LIN {X 0,Y 468.05,Z 517.764,A -85,B 0,C 180,E1 -7638.744,E2 -7638.744} C_VEL
LIN {X 0,Y 467.575,Z 526.244,A -85,B 0,C 180,E1 -7639.828,E2 -7639.828} C_VEL
LIN {X 0,Y 467.241,Z 534.525,A -85,B 0,C 180,E1 -7641.131,E2 -7641.131} C_VEL
LIN {X 0,Y 466.979,Z 541.203,A -85,B 0,C 180,E1 -7642.433,E2 -7642.433} C_VEL
LIN {X 0,Y 466.773,Z 547.316,A -85,B 0,C 180,E1 -7643.95,E2 -7643.95} C_VEL
LIN {X 0,Y 466.694,Z 551.29,A -85,B 0,C 180,E1 -7645.249,E2 -7645.249} C_VEL
LIN {X 0,Y 466.691,Z 554.227,A -85,B 0,C 180,E1 -7646.546,E2 -7646.546} C_VEL
LIN {X 0,Y 466.662,Z 555.625,A -85,B 0,C 180,E1 -7647.41,E2 -7647.41} C_VEL
LIN {X 0,Y 466.618,Z 557.234,A -85,B 0,C 180,E1 -7649.137,E2 -7649.137} C_VEL
LIN {X 0,Y 466.598,Z 557.451,A -85,B 0,C 180,E1 -7650,E2 -7650} C_VEL
LIN {X 0,Y 466.618,Z 557.236,A -85,B 0,C 180,E1 -7650.863,E2 -7650.863} C_VEL
LIN {X 0,Y 466.662,Z 555.636,A -85,B 0,C 180,E1 -7652.589,E2 -7652.589} C_VEL
LIN {X 0,Y 466.691,Z 554.239,A -85,B 0,C 180,E1 -7653.453,E2 -7653.453} C_VEL
LIN {X 0,Y 466.694,Z 551.3,A -85,B 0,C 180,E1 -7654.751,E2 -7654.751} C_VEL
LIN {X 0,Y 466.778,Z 547.322,A -85,B 0,C 180,E1 -7656.05,E2 -7656.05} C_VEL
LIN {X 0,Y 466.979,Z 541.2,A -85,B 0,C 180,E1 -7657.567,E2 -7657.567} C_VEL
LIN {X 0,Y 467.24,Z 534.511,A -85,B 0,C 180,E1 -7658.869,E2 -7658.869} C_VEL
LIN {X 0,Y 467.586,Z 526.211,A -85,B 0,C 180,E1 -7660.172,E2 -7660.172} C_VEL
LIN {X 0,Y 468.04,Z 517.699,A -85,B 0,C 180,E1 -7661.256,E2 -7661.256} C_VEL
LIN {X 0,Y 468.53,Z 507.566,A -85,B 0,C 180,E1 -7662.306,E2 -7662.306} C_VEL
LIN {X 0,Y 468.963,Z 496.77,A -85,B 0,C 180,E1 -7663.211,E2 -7663.211} C_VEL
LIN {X 0,Y 469.508,Z 485.356,A -85,B 0,C 180,E1 -7663.967,E2 -7663.967} C_VEL
LIN {X 0,Y 469.937,Z 473.595,A -85,B 0,C 180,E1 -7664.562,E2 -7664.562} C_VEL
LIN {X 0,Y 469.738,Z 468.411,A -85,B 0,C 180,E1 -7664.783,E2 -7664.783} C_VEL
LIN {X 0,Y 467.641,Z 455.017,A -85,B 0,C 180,E1 -7665.263,E2 -7665.263} C_VEL
LIN {X 0,Y 466.967,Z 450.66,A -85,B 0,C 180,E1 -7665.391,E2 -7665.391} C_VEL
LIN {X 0,Y 467.115,Z 442.772,A -85,B 0,C 180,E1 -7668.581,E2 -7668.581} C_VEL
LIN {X 0,Y 467.351,Z 435.39,A -85,B 0,C 180,E1 -7671.618,E2 -7671.618} C_VEL
LIN {X 0,Y 467.538,Z 427.589,A -85,B 0,C 180,E1 -7674.89,E2 -7674.89} C_VEL
LIN {X 0,Y 467.819,Z 419.776,A -85,B 0,C 180,E1 -7678.243,E2 -7678.243} C_VEL
LIN {X 0,Y 468.09,Z 413.208,A -85,B 0,C 180,E1 -7681.15,E2 -7681.15} C_VEL
LIN {X 0,Y 468.397,Z 406.109,A -85,B 0,C 180,E1 -7684.387,E2 -7684.387} C_VEL
LIN {X 0,Y 468.342,Z 401.978,A -85,B 0,C 180,E1 -7686.35,E2 -7686.35} C_VEL
LIN {X 0,Y 467.644,Z 397.237,A -85,B 0,C 180,E1 -7688.752,E2 -7688.752} C_VEL
LIN {X 0,Y 467.579,Z 397.243,A -85,B 0,C 180,E1 -7691.401,E2 -7691.401} C_VEL
LIN {X 0,Y 467.57,Z 397.24,A -85,B 0,C 180,E1 -7693.823,E2 -7693.823} C_VEL
LIN {X 0,Y 467.565,Z 397.242,A -85,B 0,C 180,E1 -7696.256,E2 -7696.256} C_VEL
LIN {X 0,Y 467.577,Z 397.244,A -85,B 0,C 180,E1 -7698.722,E2 -7698.722} C_VEL
LIN {X 0,Y 467.561,Z 397.242,A -85,B 0,C 180,E1 -7701.955,E2 -7701.955} C_VEL
LIN {X 0,Y 467.563,Z 397.242,A -85,B 0,C 180,E1 -7705.167,E2 -7705.167} C_VEL
LIN {X 0,Y 467.579,Z 397.242,A -85,B 0,C 180,E1 -7708.259,E2 -7708.259} C_VEL
LIN {X 0,Y 467.576,Z 397.24,A -85,B 0,C 180,E1 -7711.25,E2 -7711.25} C_VEL
LIN {X 0,Y 467.603,Z 397.239,A -85,B 0,C 180,E1 -7714.159,E2 -7714.159} C_VEL
LIN {X 0,Y 467.57,Z 397.241,A -85,B 0,C 180,E1 -7716.995,E2 -7716.995} C_VEL
LIN {X 0,Y 467.614,Z 397.237,A -85,B 0,C 180,E1 -7719.777,E2 -7719.777} C_VEL
LIN {X 0,Y 467.601,Z 397.238,A -85,B 0,C 180,E1 -7722.506,E2 -7722.506} C_VEL
LIN {X 0,Y 467.598,Z 397.239,A -85,B 0,C 180,E1 -7725.196,E2 -7725.196} C_VEL
LIN {X 0,Y 467.647,Z 397.234,A -85,B 0,C 180,E1 -7727.854,E2 -7727.854} C_VEL
LIN {X 0,Y 467.673,Z 397.23,A -85,B 0,C 180,E1 -7731.357,E2 -7731.357} C_VEL
LIN {X 0,Y 467.739,Z 397.222,A -85,B 0,C 180,E1 -7733.962,E2 -7733.962} C_VEL
LIN {X 0,Y 467.852,Z 397.208,A -85,B 0,C 180,E1 -7737.417,E2 -7737.417} C_VEL
LIN {X 0,Y 467.873,Z 397.204,A -85,B 0,C 180,E1 -7740,E2 -7740} C_VEL
LIN {X 0,Y 467.853,Z 397.207,A -85,B 0,C 180,E1 -7742.583,E2 -7742.583} C_VEL
LIN {X 0,Y 467.739,Z 397.22,A -85,B 0,C 180,E1 -7746.037,E2 -7746.037} C_VEL
LIN {X 0,Y 467.674,Z 397.232,A -85,B 0,C 180,E1 -7748.643,E2 -7748.643} C_VEL
LIN {X 0,Y 467.656,Z 397.231,A -85,B 0,C 180,E1 -7752.145,E2 -7752.145} C_VEL
LIN {X 0,Y 467.63,Z 397.233,A -85,B 0,C 180,E1 -7755.695,E2 -7755.695} C_VEL
LIN {X 0,Y 467.609,Z 397.238,A -85,B 0,C 180,E1 -7758.765,E2 -7758.765} C_VEL
LIN {X 0,Y 467.575,Z 397.24,A -85,B 0,C 180,E1 -7761.27,E2 -7761.27} C_VEL
LIN {X 0,Y 467.567,Z 397.243,A -85,B 0,C 180,E1 -7763.943,E2 -7763.943} C_VEL
LIN {X 0,Y 467.62,Z 397.235,A -85,B 0,C 180,E1 -7766.8,E2 -7766.8} C_VEL
LIN {X 0,Y 467.58,Z 397.241,A -85,B 0,C 180,E1 -7769.736,E2 -7769.736} C_VEL
LIN {X 0,Y 467.576,Z 397.24,A -85,B 0,C 180,E1 -7772.759,E2 -7772.759} C_VEL
LIN {X 0,Y 467.55,Z 397.248,A -85,B 0,C 180,E1 -7775.89,E2 -7775.89} C_VEL
LIN {X 0,Y 467.612,Z 397.235,A -85,B 0,C 180,E1 -7779.142,E2 -7779.142} C_VEL
LIN {X 0,Y 467.613,Z 397.234,A -85,B 0,C 180,E1 -7782.572,E2 -7782.572} C_VEL
LIN {X 0,Y 467.569,Z 397.24,A -85,B 0,C 180,E1 -7786.177,E2 -7786.177} C_VEL
LIN {X 0,Y 467.585,Z 397.237,A -85,B 0,C 180,E1 -7788.722,E2 -7788.722} C_VEL
LIN {X 0,Y 467.57,Z 397.245,A -85,B 0,C 180,E1 -7791.408,E2 -7791.408} C_VEL
LIN {X 0,Y 467.56,Z 397.239,A -85,B 0,C 180,E1 -7794.261,E2 -7794.261} C_VEL
LIN {X 0,Y 467.579,Z 397.245,A -85,B 0,C 180,E1 -7797.321,E2 -7797.321} C_VEL
LIN {X 0,Y 467.568,Z 397.241,A -85,B 0,C 180,E1 -7800.668,E2 -7800.668} C_VEL
LIN {X 0,Y 467.626,Z 397.238,A -85,B 0,C 180,E1 -7803.201,E2 -7803.201} C_VEL
LIN {X 0,Y 467.591,Z 397.238,A -85,B 0,C 180,E1 -7806.469,E2 -7806.469} C_VEL
LIN {X 0,Y 467.461,Z 397.258,A -85,B 0,C 180,E1 -7808.85,E2 -7808.85} C_VEL
LIN {X 0,Y 467.399,Z 398.142,A -85,B 0,C 180,E1 -7809.768,E2 -7809.768} C_VEL
LIN {X 0,Y 467.349,Z 402.042,A -85,B 0,C 180,E1 -7812.497,E2 -7812.497} C_VEL
LIN {X 0,Y 467.262,Z 406.123,A -85,B 0,C 180,E1 -7815.305,E2 -7815.305} C_VEL
LIN {X 0,Y 466.552,Z 407.238,A -85,B 0,C 180,E1 -7816.012,E2 -7816.012} C_VEL
LIN {X 0,Y 463.68,Z 409.212,A -85,B 0,C 180,E1 -7817.157,E2 -7817.157} C_VEL
LIN {X 0,Y 461.256,Z 410.811,A -85,B 0,C 180,E1 -7818.079,E2 -7818.079} C_VEL
LIN {X 0,Y 460.19,Z 411.965,A -85,B 0,C 180,E1 -7818.793,E2 -7818.793} C_VEL
LIN {X 0,Y 460.088,Z 412.332,A -85,B 0,C 180,E1 -7819.035,E2 -7819.035} C_VEL
LIN {X 0,Y 460,Z 416.903,A -85,B 0,C 180,E1 -7822.097,E2 -7822.097} C_VEL
LIN {X 0,Y 460.007,Z 419.564,A -85,B 0,C 180,E1 -7823.861,E2 -7823.861} C_VEL
LIN {X 0,Y 459.953,Z 423.574,A -85,B 0,C 180,E1 -7826.496,E2 -7826.496} C_VEL
LIN {X 0,Y 459.695,Z 426.637,A -85,B 0,C 180,E1 -7828.467,E2 -7828.467} C_VEL
LIN {X 0,Y 462.589,Z 440.592,A -85,B 0,C 180,E1 -7828.98,E2 -7828.98} C_VEL
LIN {X 0,Y 463.245,Z 445.212,A -85,B 0,C 180,E1 -7829.185,E2 -7829.185} C_VEL
LIN {X 0,Y 462.884,Z 457.387,A -85,B 0,C 180,E1 -7829.783,E2 -7829.783} C_VEL
LIN {X 0,Y 462.302,Z 469.202,A -85,B 0,C 180,E1 -7830.545,E2 -7830.545} C_VEL
LIN {X 0,Y 461.851,Z 479.727,A -85,B 0,C 180,E1 -7831.417,E2 -7831.417} C_VEL
LIN {X 0,Y 461.333,Z 489.381,A -85,B 0,C 180,E1 -7832.401,E2 -7832.401} C_VEL
LIN {X 0,Y 460.819,Z 498.195,A -85,B 0,C 180,E1 -7833.498,E2 -7833.498} C_VEL
LIN {X 0,Y 460.377,Z 506.8,A -85,B 0,C 180,E1 -7834.816,E2 -7834.816} C_VEL
LIN {X 0,Y 460.156,Z 513.662,A -85,B 0,C 180,E1 -7836.137,E2 -7836.137} C_VEL
LIN {X 0,Y 459.923,Z 519.186,A -85,B 0,C 180,E1 -7837.463,E2 -7837.463} C_VEL
LIN {X 0,Y 459.711,Z 523.535,A -85,B 0,C 180,E1 -7838.794,E2 -7838.794} C_VEL
LIN {X 0,Y 459.612,Z 525.839,A -85,B 0,C 180,E1 -7839.683,E2 -7839.683} C_VEL
LIN {X 0,Y 459.606,Z 527.696,A -85,B 0,C 180,E1 -7840.573,E2 -7840.573} C_VEL
LIN {X 0,Y 459.566,Z 529.559,A -85,B 0,C 180,E1 -7841.838,E2 -7841.838} C_VEL
LIN {X 0,Y 459.439,Z 530.67,A -85,B 0,C 180,E1 -7843.265,E2 -7843.265} C_VEL
LIN {X 0,Y 459.437,Z 530.824,A -85,B 0,C 180,E1 -7844.167,E2 -7844.167} C_VEL
LIN {X 0,Y 459.496,Z 530.297,A -85,B 0,C 180,E1 -7845.51,E2 -7845.51} C_VEL
LIN {X 0,Y 459.465,Z 528.774,A -85,B 0,C 180,E1 -7846.895,E2 -7846.895} C_VEL
LIN {X 0,Y 459.645,Z 525.549,A -85,B 0,C 180,E1 -7848.561,E2 -7848.561} C_VEL
LIN {X 0,Y 459.816,Z 521.139,A -85,B 0,C 180,E1 -7850.114,E2 -7850.114} C_VEL
LIN {X 0,Y 460.065,Z 515.868,A -85,B 0,C 180,E1 -7851.507,E2 -7851.507} C_VEL
LIN {X 0,Y 460.391,Z 509.082,A -85,B 0,C 180,E1 -7852.908,E2 -7852.908} C_VEL
LIN {X 0,Y 460.803,Z 500.493,A -85,B 0,C 180,E1 -7854.317,E2 -7854.317} C_VEL
LIN {X 0,Y 461.28,Z 491.756,A -85,B 0,C 180,E1 -7855.473,E2 -7855.473} C_VEL
LIN {X 0,Y 461.797,Z 481.616,A -85,B 0,C 180,E1 -7856.554,E2 -7856.554} C_VEL
LIN {X 0,Y 462.412,Z 470.625,A -85,B 0,C 180,E1 -7857.494,E2 -7857.494} C_VEL
LIN {X 0,Y 462.852,Z 460.595,A -85,B 0,C 180,E1 -7858.181,E2 -7858.181} C_VEL
LIN {X 0,Y 463.292,Z 448.73,A -85,B 0,C 180,E1 -7858.817,E2 -7858.817} C_VEL
LIN {X 0,Y 463.261,Z 443.626,A -85,B 0,C 180,E1 -7859.042,E2 -7859.042} C_VEL
LIN {X 0,Y 460.731,Z 431.182,A -85,B 0,C 180,E1 -7859.558,E2 -7859.558} C_VEL
LIN {X 0,Y 459.714,Z 426.771,A -85,B 0,C 180,E1 -7859.711,E2 -7859.711} C_VEL
LIN {X 0,Y 459.836,Z 422.121,A -85,B 0,C 180,E1 -7862.796,E2 -7862.796} C_VEL
LIN {X 0,Y 459.944,Z 417.5,A -85,B 0,C 180,E1 -7865.919,E2 -7865.919} C_VEL
LIN {X 0,Y 460.079,Z 413.289,A -85,B 0,C 180,E1 -7868.826,E2 -7868.826} C_VEL
LIN {X 0,Y 460.181,Z 409.438,A -85,B 0,C 180,E1 -7871.553,E2 -7871.553} C_VEL
LIN {X 0,Y 460.298,Z 405.231,A -85,B 0,C 180,E1 -7874.615,E2 -7874.615} C_VEL
LIN {X 0,Y 460.461,Z 400.928,A -85,B 0,C 180,E1 -7877.812,E2 -7877.812} C_VEL
LIN {X 0,Y 460.444,Z 398.134,A -85,B 0,C 180,E1 -7880.129,E2 -7880.129} C_VEL
LIN {X 0,Y 460.496,Z 398.129,A -85,B 0,C 180,E1 -7882.523,E2 -7882.523} C_VEL
LIN {X 0,Y 460.543,Z 398.121,A -85,B 0,C 180,E1 -7885.624,E2 -7885.624} C_VEL
LIN {X 0,Y 460.531,Z 398.12,A -85,B 0,C 180,E1 -7888.744,E2 -7888.744} C_VEL
LIN {X 0,Y 460.553,Z 398.117,A -85,B 0,C 180,E1 -7891.767,E2 -7891.767} C_VEL
LIN {X 0,Y 460.554,Z 398.117,A -85,B 0,C 180,E1 -7894.705,E2 -7894.705} C_VEL
LIN {X 0,Y 460.505,Z 398.122,A -85,B 0,C 180,E1 -7897.571,E2 -7897.571} C_VEL
LIN {X 0,Y 460.562,Z 398.116,A -85,B 0,C 180,E1 -7900.384,E2 -7900.384} C_VEL
LIN {X 0,Y 460.559,Z 398.117,A -85,B 0,C 180,E1 -7903.146,E2 -7903.146} C_VEL
LIN {X 0,Y 460.548,Z 398.118,A -85,B 0,C 180,E1 -7905.868,E2 -7905.868} C_VEL
LIN {X 0,Y 460.607,Z 398.109,A -85,B 0,C 180,E1 -7908.559,E2 -7908.559} C_VEL
LIN {X 0,Y 460.688,Z 398.103,A -85,B 0,C 180,E1 -7912.109,E2 -7912.109} C_VEL
LIN {X 0,Y 460.691,Z 398.1,A -85,B 0,C 180,E1 -7914.748,E2 -7914.748} C_VEL
LIN {X 0,Y 460.819,Z 398.082,A -85,B 0,C 180,E1 -7917.378,E2 -7917.378} C_VEL
LIN {X 0,Y 460.846,Z 398.08,A -85,B 0,C 180,E1 -7920,E2 -7920} C_VEL
LIN {X 0,Y 460.819,Z 398.086,A -85,B 0,C 180,E1 -7922.623,E2 -7922.623} C_VEL
LIN {X 0,Y 460.704,Z 398.097,A -85,B 0,C 180,E1 -7926.13,E2 -7926.13} C_VEL
LIN {X 0,Y 460.623,Z 398.109,A -85,B 0,C 180,E1 -7928.776,E2 -7928.776} C_VEL
LIN {X 0,Y 460.628,Z 398.107,A -85,B 0,C 180,E1 -7932.457,E2 -7932.457} C_VEL
LIN {X 0,Y 460.616,Z 398.113,A -85,B 0,C 180,E1 -7936.008,E2 -7936.008} C_VEL
LIN {X 0,Y 460.564,Z 398.116,A -85,B 0,C 180,E1 -7939.616,E2 -7939.616} C_VEL
LIN {X 0,Y 460.507,Z 398.124,A -85,B 0,C 180,E1 -7942.429,E2 -7942.429} C_VEL
LIN {X 0,Y 460.564,Z 398.116,A -85,B 0,C 180,E1 -7945.803,E2 -7945.803} C_VEL
LIN {X 0,Y 460.554,Z 398.118,A -85,B 0,C 180,E1 -7948.233,E2 -7948.233} C_VEL
LIN {X 0,Y 460.521,Z 398.122,A -85,B 0,C 180,E1 -7951.284,E2 -7951.284} C_VEL
LIN {X 0,Y 460.53,Z 398.119,A -85,B 0,C 180,E1 -7954.507,E2 -7954.507} C_VEL
LIN {X 0,Y 460.525,Z 398.116,A -85,B 0,C 180,E1 -7957.621,E2 -7957.621} C_VEL
LIN {X 0,Y 460.539,Z 398.119,A -85,B 0,C 180,E1 -7960.27,E2 -7960.27} C_VEL
LIN {X 0,Y 460.498,Z 398.125,A -85,B 0,C 180,E1 -7963.376,E2 -7963.376} C_VEL
LIN {X 0,Y 460.507,Z 398.123,A -85,B 0,C 180,E1 -7966.626,E2 -7966.626} C_VEL
LIN {X 0,Y 460.556,Z 398.119,A -85,B 0,C 180,E1 -7969.937,E2 -7969.937} C_VEL
LIN {X 0,Y 461.273,Z 402.381,A -85,B 0,C 180,E1 -7972.451,E2 -7972.451} C_VEL
LIN {X 0,Y 461.655,Z 406.549,A -85,B 0,C 180,E1 -7974.656,E2 -7974.656} C_VEL
LIN {X 0,Y 461.413,Z 411.029,A -85,B 0,C 180,E1 -7976.902,E2 -7976.902} C_VEL
LIN {X 0,Y 461.136,Z 417.074,A -85,B 0,C 180,E1 -7979.806,E2 -7979.806} C_VEL
LIN {X 0,Y 460.713,Z 423.504,A -85,B 0,C 180,E1 -7982.766,E2 -7982.766} C_VEL
LIN {X 0,Y 460.467,Z 429.999,A -85,B 0,C 180,E1 -7985.664,E2 -7985.664} C_VEL
LIN {X 0,Y 460.277,Z 436.882,A -85,B 0,C 180,E1 -7988.657,E2 -7988.657} C_VEL
LIN {X 0,Y 460.03,Z 444.198,A -85,B 0,C 180,E1 -7991.749,E2 -7991.749} C_VEL
LIN {X 0,Y 459.886,Z 450.374,A -85,B 0,C 180,E1 -7994.317,E2 -7994.317} C_VEL
LIN {X 0,Y 462.057,Z 463.442,A -85,B 0,C 180,E1 -7994.748,E2 -7994.748} C_VEL
LIN {X 0,Y 463.163,Z 472.924,A -85,B 0,C 180,E1 -7995.164,E2 -7995.164} C_VEL
LIN {X 0,Y 462.724,Z 483.778,A -85,B 0,C 180,E1 -7995.711,E2 -7995.711} C_VEL
LIN {X 0,Y 462.174,Z 495.488,A -85,B 0,C 180,E1 -7996.479,E2 -7996.479} C_VEL
LIN {X 0,Y 461.704,Z 505.916,A -85,B 0,C 180,E1 -7997.348,E2 -7997.348} C_VEL
LIN {X 0,Y 461.199,Z 515.71,A -85,B 0,C 180,E1 -7998.351,E2 -7998.351} C_VEL
LIN {X 0,Y 460.622,Z 524.523,A -85,B 0,C 180,E1 -7999.45,E2 -7999.45} C_VEL
LIN {X 0,Y 460.241,Z 533.123,A -85,B 0,C 180,E1 -8000.774,E2 -8000.774} C_VEL
LIN {X 0,Y 459.952,Z 540.009,A -85,B 0,C 180,E1 -8002.096,E2 -8002.096} C_VEL
LIN {X 0,Y 459.715,Z 546.095,A -85,B 0,C 180,E1 -8003.569,E2 -8003.569} C_VEL
LIN {X 0,Y 459.622,Z 551.095,A -85,B 0,C 180,E1 -8005.176,E2 -8005.176} C_VEL
LIN {X 0,Y 459.586,Z 554.03,A -85,B 0,C 180,E1 -8006.493,E2 -8006.493} C_VEL
LIN {X 0,Y 459.585,Z 555.426,A -85,B 0,C 180,E1 -8007.37,E2 -8007.37} C_VEL
LIN {X 0,Y 459.522,Z 557.032,A -85,B 0,C 180,E1 -8009.124,E2 -8009.124} C_VEL
LIN {X 0,Y 459.53,Z 557.248,A -85,B 0,C 180,E1 -8010,E2 -8010} C_VEL
LIN {X 0,Y 459.521,Z 557.03,A -85,B 0,C 180,E1 -8010.876,E2 -8010.876} C_VEL
LIN {X 0,Y 459.585,Z 555.427,A -85,B 0,C 180,E1 -8012.629,E2 -8012.629} C_VEL
LIN {X 0,Y 459.586,Z 554.026,A -85,B 0,C 180,E1 -8013.507,E2 -8013.507} C_VEL
LIN {X 0,Y 459.622,Z 551.085,A -85,B 0,C 180,E1 -8014.824,E2 -8014.824} C_VEL
LIN {X 0,Y 459.714,Z 546.066,A -85,B 0,C 180,E1 -8016.431,E2 -8016.431} C_VEL
LIN {X 0,Y 459.951,Z 539.96,A -85,B 0,C 180,E1 -8017.904,E2 -8017.904} C_VEL
LIN {X 0,Y 460.24,Z 533.036,A -85,B 0,C 180,E1 -8019.226,E2 -8019.226} C_VEL
LIN {X 0,Y 460.629,Z 524.356,A -85,B 0,C 180,E1 -8020.549,E2 -8020.549} C_VEL
LIN {X 0,Y 461.137,Z 515.46,A -85,B 0,C 180,E1 -8021.65,E2 -8021.65} C_VEL
LIN {X 0,Y 461.686,Z 505.699,A -85,B 0,C 180,E1 -8022.639,E2 -8022.639} C_VEL
LIN {X 0,Y 462.133,Z 494.977,A -85,B 0,C 180,E1 -8023.522,E2 -8023.522} C_VEL
LIN {X 0,Y 462.646,Z 482.967,A -85,B 0,C 180,E1 -8024.291,E2 -8024.291} C_VEL
LIN {X 0,Y 463.091,Z 471.765,A -85,B 0,C 180,E1 -8024.838,E2 -8024.838} C_VEL
LIN {X 0,Y 461.183,Z 458.423,A -85,B 0,C 180,E1 -8025.376,E2 -8025.376} C_VEL
LIN {X 0,Y 459.881,Z 450.497,A -85,B 0,C 180,E1 -8025.612,E2 -8025.612} C_VEL
LIN {X 0,Y 460.053,Z 442.965,A -85,B 0,C 180,E1 -8028.711,E2 -8028.711} C_VEL
LIN {X 0,Y 460.301,Z 435.181,A -85,B 0,C 180,E1 -8031.966,E2 -8031.966} C_VEL
LIN {X 0,Y 460.523,Z 427.377,A -85,B 0,C 180,E1 -8035.296,E2 -8035.296} C_VEL
LIN {X 0,Y 460.837,Z 419.593,A -85,B 0,C 180,E1 -8038.71,E2 -8038.71} C_VEL
LIN {X 0,Y 461.094,Z 413.614,A -85,B 0,C 180,E1 -8041.399,E2 -8041.399} C_VEL
LIN {X 0,Y 461.399,Z 406.578,A -85,B 0,C 180,E1 -8044.661,E2 -8044.661} C_VEL
LIN {X 0,Y 461.297,Z 402.887,A -85,B 0,C 180,E1 -8046.453,E2 -8046.453} C_VEL
LIN {X 0,Y 460.604,Z 398.114,A -85,B 0,C 180,E1 -8048.906,E2 -8048.906} C_VEL
LIN {X 0,Y 460.523,Z 398.12,A -85,B 0,C 180,E1 -8052.18,E2 -8052.18} C_VEL
LIN {X 0,Y 460.517,Z 398.12,A -85,B 0,C 180,E1 -8055.411,E2 -8055.411} C_VEL
LIN {X 0,Y 460.53,Z 398.119,A -85,B 0,C 180,E1 -8058.396,E2 -8058.396} C_VEL
LIN {X 0,Y 460.521,Z 398.119,A -85,B 0,C 180,E1 -8061.266,E2 -8061.266} C_VEL
LIN {X 0,Y 460.508,Z 398.124,A -85,B 0,C 180,E1 -8064.554,E2 -8064.554} C_VEL
LIN {X 0,Y 460.526,Z 398.119,A -85,B 0,C 180,E1 -8067.715,E2 -8067.715} C_VEL
LIN {X 0,Y 460.541,Z 398.119,A -85,B 0,C 180,E1 -8070.769,E2 -8070.769} C_VEL
LIN {X 0,Y 460.556,Z 398.116,A -85,B 0,C 180,E1 -8073.734,E2 -8073.734} C_VEL
LIN {X 0,Y 460.539,Z 398.119,A -85,B 0,C 180,E1 -8076.623,E2 -8076.623} C_VEL
LIN {X 0,Y 460.543,Z 398.118,A -85,B 0,C 180,E1 -8079.452,E2 -8079.452} C_VEL
LIN {X 0,Y 460.551,Z 398.119,A -85,B 0,C 180,E1 -8082.23,E2 -8082.23} C_VEL
LIN {X 0,Y 460.557,Z 398.115,A -85,B 0,C 180,E1 -8084.964,E2 -8084.964} C_VEL
LIN {X 0,Y 460.602,Z 398.109,A -85,B 0,C 180,E1 -8088.559,E2 -8088.559} C_VEL
LIN {X 0,Y 460.686,Z 398.1,A -85,B 0,C 180,E1 -8092.108,E2 -8092.108} C_VEL
LIN {X 0,Y 460.694,Z 398.099,A -85,B 0,C 180,E1 -8094.748,E2 -8094.748} C_VEL
LIN {X 0,Y 460.817,Z 398.084,A -85,B 0,C 180,E1 -8097.377,E2 -8097.377} C_VEL
LIN {X 0,Y 460.844,Z 398.08,A -85,B 0,C 180,E1 -8100,E2 -8100} C_VEL
LIN {X 0,Y 460.818,Z 398.084,A -85,B 0,C 180,E1 -8102.622,E2 -8102.622} C_VEL
LIN {X 0,Y 460.704,Z 398.097,A -85,B 0,C 180,E1 -8106.13,E2 -8106.13} C_VEL
LIN {X 0,Y 460.621,Z 398.11,A -85,B 0,C 180,E1 -8108.776,E2 -8108.776} C_VEL
LIN {X 0,Y 460.625,Z 398.109,A -85,B 0,C 180,E1 -8112.457,E2 -8112.457} C_VEL
LIN {X 0,Y 460.591,Z 398.111,A -85,B 0,C 180,E1 -8115.998,E2 -8115.998} C_VEL
LIN {X 0,Y 460.562,Z 398.115,A -85,B 0,C 180,E1 -8118.902,E2 -8118.902} C_VEL
LIN {X 0,Y 460.51,Z 398.12,A -85,B 0,C 180,E1 -8121.486,E2 -8121.486} C_VEL
LIN {X 0,Y 460.536,Z 398.121,A -85,B 0,C 180,E1 -8124.332,E2 -8124.332} C_VEL
LIN {X 0,Y 460.576,Z 398.112,A -85,B 0,C 180,E1 -8127.243,E2 -8127.243} C_VEL
LIN {X 0,Y 460.52,Z 398.122,A -85,B 0,C 180,E1 -8130.239,E2 -8130.239} C_VEL
LIN {X 0,Y 460.522,Z 398.118,A -85,B 0,C 180,E1 -8133.325,E2 -8133.325} C_VEL
LIN {X 0,Y 460.473,Z 398.125,A -85,B 0,C 180,E1 -8136.53,E2 -8136.53} C_VEL
LIN {X 0,Y 460.572,Z 398.117,A -85,B 0,C 180,E1 -8139.858,E2 -8139.858} C_VEL
LIN {X 0,Y 460.537,Z 398.115,A -85,B 0,C 180,E1 -8142.905,E2 -8142.905} C_VEL
LIN {X 0,Y 460.519,Z 398.122,A -85,B 0,C 180,E1 -8145.829,E2 -8145.829} C_VEL
LIN {X 0,Y 460.538,Z 398.116,A -85,B 0,C 180,E1 -8148.991,E2 -8148.991} C_VEL
LIN {X 0,Y 460.54,Z 398.119,A -85,B 0,C 180,E1 -8151.269,E2 -8151.269} C_VEL
LIN {X 0,Y 460.51,Z 398.118,A -85,B 0,C 180,E1 -8154.555,E2 -8154.555} C_VEL
LIN {X 0,Y 460.529,Z 398.118,A -85,B 0,C 180,E1 -8157.716,E2 -8157.716} C_VEL
LIN {X 0,Y 460.538,Z 398.117,A -85,B 0,C 180,E1 -8160.77,E2 -8160.77} C_VEL
LIN {X 0,Y 460.567,Z 398.112,A -85,B 0,C 180,E1 -8163.736,E2 -8163.736} C_VEL
LIN {X 0,Y 460.543,Z 398.117,A -85,B 0,C 180,E1 -8166.625,E2 -8166.625} C_VEL
LIN {X 0,Y 460.443,Z 398.13,A -85,B 0,C 180,E1 -8168.603,E2 -8168.603} C_VEL
LIN {X 0,Y 460.344,Z 398.538,A -85,B 0,C 180,E1 -8169.444,E2 -8169.444} C_VEL
LIN {X 0,Y 460.298,Z 402.449,A -85,B 0,C 180,E1 -8172.22,E2 -8172.22} C_VEL
LIN {X 0,Y 460.223,Z 406.365,A -85,B 0,C 180,E1 -8174.954,E2 -8174.954} C_VEL
LIN {X 0,Y 460.2,Z 410.499,A -85,B 0,C 180,E1 -8177.791,E2 -8177.791} C_VEL
LIN {X 0,Y 460.088,Z 412.332,A -85,B 0,C 180,E1 -8179.035,E2 -8179.035} C_VEL
LIN {X 0,Y 459.366,Z 413.461,A -85,B 0,C 180,E1 -8179.752,E2 -8179.752} C_VEL
LIN {X 0,Y 456.451,Z 415.46,A -85,B 0,C 180,E1 -8180.911,E2 -8180.911} C_VEL
LIN {X 0,Y 454.033,Z 417.074,A -85,B 0,C 180,E1 -8181.845,E2 -8181.845} C_VEL
LIN {X 0,Y 453.028,Z 418.243,A -85,B 0,C 180,E1 -8182.57,E2 -8182.57} C_VEL
LIN {X 0,Y 452.962,Z 418.616,A -85,B 0,C 180,E1 -8182.815,E2 -8182.815} C_VEL
LIN {X 0,Y 452.933,Z 422.711,A -85,B 0,C 180,E1 -8185.551,E2 -8185.551} C_VEL
LIN {X 0,Y 452.681,Z 427.047,A -85,B 0,C 180,E1 -8188.249,E2 -8188.249} C_VEL
LIN {X 0,Y 455.494,Z 440.42,A -85,B 0,C 180,E1 -8188.743,E2 -8188.743} C_VEL
LIN {X 0,Y 456.355,Z 446.236,A -85,B 0,C 180,E1 -8189.007,E2 -8189.007} C_VEL
LIN {X 0,Y 455.91,Z 459.209,A -85,B 0,C 180,E1 -8189.669,E2 -8189.669} C_VEL
LIN {X 0,Y 455.335,Z 470.579,A -85,B 0,C 180,E1 -8190.442,E2 -8190.442} C_VEL
LIN {X 0,Y 454.767,Z 482.07,A -85,B 0,C 180,E1 -8191.439,E2 -8191.439} C_VEL
LIN {X 0,Y 454.263,Z 491.361,A -85,B 0,C 180,E1 -8192.439,E2 -8192.439} C_VEL
LIN {X 0,Y 453.733,Z 499.864,A -85,B 0,C 180,E1 -8193.552,E2 -8193.552} C_VEL
LIN {X 0,Y 453.296,Z 508.128,A -85,B 0,C 180,E1 -8194.892,E2 -8194.892} C_VEL
LIN {X 0,Y 453.077,Z 514.787,A -85,B 0,C 180,E1 -8196.234,E2 -8196.234} C_VEL
LIN {X 0,Y 452.821,Z 520.132,A -85,B 0,C 180,E1 -8197.581,E2 -8197.581} C_VEL
LIN {X 0,Y 452.602,Z 524.313,A -85,B 0,C 180,E1 -8198.933,E2 -8198.933} C_VEL
LIN {X 0,Y 452.512,Z 526.522,A -85,B 0,C 180,E1 -8199.837,E2 -8199.837} C_VEL
LIN {X 0,Y 452.497,Z 528.24,A -85,B 0,C 180,E1 -8200.741,E2 -8200.741} C_VEL
LIN {X 0,Y 452.466,Z 529.848,A -85,B 0,C 180,E1 -8201.887,E2 -8201.887} C_VEL
LIN {X 0,Y 452.349,Z 530.941,A -85,B 0,C 180,E1 -8203.477,E2 -8203.477} C_VEL
LIN {X 0,Y 452.347,Z 530.991,A -85,B 0,C 180,E1 -8204.394,E2 -8204.394} C_VEL
LIN {X 0,Y 452.398,Z 530.457,A -85,B 0,C 180,E1 -8205.599,E2 -8205.599} C_VEL
LIN {X 0,Y 452.391,Z 528.636,A -85,B 0,C 180,E1 -8207.168,E2 -8207.168} C_VEL
LIN {X 0,Y 452.562,Z 525.661,A -85,B 0,C 180,E1 -8208.686,E2 -8208.686} C_VEL
LIN {X 0,Y 452.736,Z 522.148,A -85,B 0,C 180,E1 -8209.969,E2 -8209.969} C_VEL
LIN {X 0,Y 452.995,Z 516.913,A -85,B 0,C 180,E1 -8211.429,E2 -8211.429} C_VEL
LIN {X 0,Y 453.282,Z 510.628,A -85,B 0,C 180,E1 -8212.806,E2 -8212.806} C_VEL
LIN {X 0,Y 453.667,Z 503.761,A -85,B 0,C 180,E1 -8214.021,E2 -8214.021} C_VEL
LIN {X 0,Y 454.13,Z 495.736,A -85,B 0,C 180,E1 -8215.187,E2 -8215.187} C_VEL
LIN {X 0,Y 454.676,Z 485.458,A -85,B 0,C 180,E1 -8216.396,E2 -8216.396} C_VEL
LIN {X 0,Y 455.366,Z 474.141,A -85,B 0,C 180,E1 -8217.457,E2 -8217.457} C_VEL
LIN {X 0,Y 455.912,Z 462.722,A -85,B 0,C 180,E1 -8218.295,E2 -8218.295} C_VEL
LIN {X 0,Y 456.401,Z 450.91,A -85,B 0,C 180,E1 -8218.966,E2 -8218.966} C_VEL
LIN {X 0,Y 456.499,Z 445.05,A -85,B 0,C 180,E1 -8219.236,E2 -8219.236} C_VEL
LIN {X 0,Y 453.984,Z 432.627,A -85,B 0,C 180,E1 -8219.784,E2 -8219.784} C_VEL
LIN {X 0,Y 452.671,Z 426.954,A -85,B 0,C 180,E1 -8219.994,E2 -8219.994} C_VEL
LIN {X 0,Y 452.772,Z 422.418,A -85,B 0,C 180,E1 -8223.05,E2 -8223.05} C_VEL
LIN {X 0,Y 452.892,Z 417.827,A -85,B 0,C 180,E1 -8226.202,E2 -8226.202} C_VEL
LIN {X 0,Y 453.031,Z 413.16,A -85,B 0,C 180,E1 -8229.497,E2 -8229.497} C_VEL
LIN {X 0,Y 453.137,Z 409.826,A -85,B 0,C 180,E1 -8231.887,E2 -8231.887} C_VEL
LIN {X 0,Y 453.246,Z 406.293,A -85,B 0,C 180,E1 -8234.498,E2 -8234.498} C_VEL
LIN {X 0,Y 453.383,Z 402.974,A -85,B 0,C 180,E1 -8236.996,E2 -8236.996} C_VEL
LIN {X 0,Y 453.458,Z 399.859,A -85,B 0,C 180,E1 -8239.413,E2 -8239.413} C_VEL
LIN {X 0,Y 453.421,Z 399.009,A -85,B 0,C 180,E1 -8240.804,E2 -8240.804} C_VEL
LIN {X 0,Y 453.453,Z 399.007,A -85,B 0,C 180,E1 -8243.917,E2 -8243.917} C_VEL
LIN {X 0,Y 453.478,Z 399,A -85,B 0,C 180,E1 -8247.151,E2 -8247.151} C_VEL
LIN {X 0,Y 453.509,Z 398.994,A -85,B 0,C 180,E1 -8250.271,E2 -8250.271} C_VEL
LIN {X 0,Y 453.508,Z 398.994,A -85,B 0,C 180,E1 -8253.294,E2 -8253.294} C_VEL
LIN {X 0,Y 453.497,Z 398.995,A -85,B 0,C 180,E1 -8256.239,E2 -8256.239} C_VEL
LIN {X 0,Y 453.476,Z 398.999,A -85,B 0,C 180,E1 -8259.117,E2 -8259.117} C_VEL
LIN {X 0,Y 453.505,Z 398.995,A -85,B 0,C 180,E1 -8261.944,E2 -8261.944} C_VEL
LIN {X 0,Y 453.533,Z 398.993,A -85,B 0,C 180,E1 -8264.726,E2 -8264.726} C_VEL
LIN {X 0,Y 453.555,Z 398.987,A -85,B 0,C 180,E1 -8268.379,E2 -8268.379} C_VEL
LIN {X 0,Y 453.645,Z 398.979,A -85,B 0,C 180,E1 -8271.985,E2 -8271.985} C_VEL
LIN {X 0,Y 453.665,Z 398.975,A -85,B 0,C 180,E1 -8274.667,E2 -8274.667} C_VEL
LIN {X 0,Y 453.759,Z 398.962,A -85,B 0,C 180,E1 -8277.337,E2 -8277.337} C_VEL
LIN {X 0,Y 453.817,Z 398.956,A -85,B 0,C 180,E1 -8280,E2 -8280} C_VEL
LIN {X 0,Y 453.76,Z 398.965,A -85,B 0,C 180,E1 -8282.663,E2 -8282.663} C_VEL
LIN {X 0,Y 453.671,Z 398.973,A -85,B 0,C 180,E1 -8286.226,E2 -8286.226} C_VEL
LIN {X 0,Y 453.587,Z 398.985,A -85,B 0,C 180,E1 -8288.914,E2 -8288.914} C_VEL
LIN {X 0,Y 453.596,Z 398.983,A -85,B 0,C 180,E1 -8292.551,E2 -8292.551} C_VEL
LIN {X 0,Y 453.551,Z 398.992,A -85,B 0,C 180,E1 -8296.196,E2 -8296.196} C_VEL
LIN {X 0,Y 453.515,Z 398.997,A -85,B 0,C 180,E1 -8299.041,E2 -8299.041} C_VEL
LIN {X 0,Y 453.472,Z 399.003,A -85,B 0,C 180,E1 -8301.837,E2 -8301.837} C_VEL
LIN {X 0,Y 453.51,Z 398.997,A -85,B 0,C 180,E1 -8304.735,E2 -8304.735} C_VEL
LIN {X 0,Y 453.534,Z 398.995,A -85,B 0,C 180,E1 -8307.962,E2 -8307.962} C_VEL
LIN {X 0,Y 453.479,Z 399.001,A -85,B 0,C 180,E1 -8310.76,E2 -8310.76} C_VEL
LIN {X 0,Y 453.474,Z 399.001,A -85,B 0,C 180,E1 -8313.913,E2 -8313.913} C_VEL
LIN {X 0,Y 453.467,Z 398.997,A -85,B 0,C 180,E1 -8317.189,E2 -8317.189} C_VEL
LIN {X 0,Y 453.487,Z 398.995,A -85,B 0,C 180,E1 -8319.45,E2 -8319.45} C_VEL
LIN {X 0,Y 453.474,Z 398.999,A -85,B 0,C 180,E1 -8321.935,E2 -8321.935} C_VEL
LIN {X 0,Y 453.489,Z 398.998,A -85,B 0,C 180,E1 -8325.471,E2 -8325.471} C_VEL
LIN {X 0,Y 453.48,Z 399,A -85,B 0,C 180,E1 -8328.21,E2 -8328.21} C_VEL
LIN {X 0,Y 453.541,Z 399.099,A -85,B 0,C 180,E1 -8329.773,E2 -8329.773} C_VEL
LIN {X 0,Y 454.433,Z 404.491,A -85,B 0,C 180,E1 -8332.905,E2 -8332.905} C_VEL
LIN {X 0,Y 454.629,Z 408.657,A -85,B 0,C 180,E1 -8335.113,E2 -8335.113} C_VEL
LIN {X 0,Y 454.316,Z 413.892,A -85,B 0,C 180,E1 -8337.745,E2 -8337.745} C_VEL
LIN {X 0,Y 453.966,Z 420.259,A -85,B 0,C 180,E1 -8340.813,E2 -8340.813} C_VEL
LIN {X 0,Y 453.566,Z 427.769,A -85,B 0,C 180,E1 -8344.288,E2 -8344.288} C_VEL
LIN {X 0,Y 453.26,Z 435.346,A -85,B 0,C 180,E1 -8347.674,E2 -8347.674} C_VEL
LIN {X 0,Y 453.062,Z 441.883,A -85,B 0,C 180,E1 -8350.518,E2 -8350.518} C_VEL
LIN {X 0,Y 452.854,Z 450.146,A -85,B 0,C 180,E1 -8354.031,E2 -8354.031} C_VEL
LIN {X 0,Y 455.218,Z 464.161,A -85,B 0,C 180,E1 -8354.528,E2 -8354.528} C_VEL
LIN {X 0,Y 456.301,Z 473.111,A -85,B 0,C 180,E1 -8354.935,E2 -8354.935} C_VEL
LIN {X 0,Y 455.747,Z 485.689,A -85,B 0,C 180,E1 -8355.602,E2 -8355.602} C_VEL
LIN {X 0,Y 455.058,Z 498.313,A -85,B 0,C 180,E1 -8356.491,E2 -8356.491} C_VEL
LIN {X 0,Y 454.531,Z 509.434,A -85,B 0,C 180,E1 -8357.498,E2 -8357.498} C_VEL
LIN {X 0,Y 453.971,Z 519.339,A -85,B 0,C 180,E1 -8358.616,E2 -8358.616} C_VEL
LIN {X 0,Y 453.47,Z 527.47,A -85,B 0,C 180,E1 -8359.733,E2 -8359.733} C_VEL
LIN {X 0,Y 453.099,Z 535.461,A -85,B 0,C 180,E1 -8361.077,E2 -8361.077} C_VEL
LIN {X 0,Y 452.817,Z 541.865,A -85,B 0,C 180,E1 -8362.419,E2 -8362.419} C_VEL
LIN {X 0,Y 452.605,Z 546.958,A -85,B 0,C 180,E1 -8363.76,E2 -8363.76} C_VEL
LIN {X 0,Y 452.55,Z 550.917,A -85,B 0,C 180,E1 -8365.1,E2 -8365.1} C_VEL
LIN {X 0,Y 452.482,Z 553.842,A -85,B 0,C 180,E1 -8366.438,E2 -8366.438} C_VEL
LIN {X 0,Y 452.508,Z 555.234,A -85,B 0,C 180,E1 -8367.329,E2 -8367.329} C_VEL
LIN {X 0,Y 452.428,Z 556.832,A -85,B 0,C 180,E1 -8369.11,E2 -8369.11} C_VEL
LIN {X 0,Y 452.434,Z 557.043,A -85,B 0,C 180,E1 -8370,E2 -8370} C_VEL
LIN {X 0,Y 452.437,Z 556.21,A -85,B 0,C 180,E1 -8371.78,E2 -8371.78} C_VEL
LIN {X 0,Y 452.508,Z 555.212,A -85,B 0,C 180,E1 -8372.67,E2 -8372.67} C_VEL
LIN {X 0,Y 452.483,Z 553.804,A -85,B 0,C 180,E1 -8373.562,E2 -8373.562} C_VEL
LIN {X 0,Y 452.55,Z 550.856,A -85,B 0,C 180,E1 -8374.9,E2 -8374.9} C_VEL
LIN {X 0,Y 452.629,Z 546.239,A -85,B 0,C 180,E1 -8376.416,E2 -8376.416} C_VEL
LIN {X 0,Y 452.893,Z 539.696,A -85,B 0,C 180,E1 -8378.028,E2 -8378.028} C_VEL
LIN {X 0,Y 453.208,Z 532.753,A -85,B 0,C 180,E1 -8379.371,E2 -8379.371} C_VEL
LIN {X 0,Y 453.624,Z 524.048,A -85,B 0,C 180,E1 -8380.714,E2 -8380.714} C_VEL
LIN {X 0,Y 454.16,Z 515.131,A -85,B 0,C 180,E1 -8381.831,E2 -8381.831} C_VEL
LIN {X 0,Y 454.683,Z 504.585,A -85,B 0,C 180,E1 -8382.909,E2 -8382.909} C_VEL
LIN {X 0,Y 455.206,Z 494.58,A -85,B 0,C 180,E1 -8383.731,E2 -8383.731} C_VEL
LIN {X 0,Y 455.728,Z 482.509,A -85,B 0,C 180,E1 -8384.512,E2 -8384.512} C_VEL
LIN {X 0,Y 456.03,Z 471.217,A -85,B 0,C 180,E1 -8385.073,E2 -8385.073} C_VEL
LIN {X 0,Y 454.048,Z 457.919,A -85,B 0,C 180,E1 -8385.615,E2 -8385.615} C_VEL
LIN {X 0,Y 452.833,Z 450.293,A -85,B 0,C 180,E1 -8385.847,E2 -8385.847} C_VEL
LIN {X 0,Y 452.99,Z 442.73,A -85,B 0,C 180,E1 -8389.014,E2 -8389.014} C_VEL
LIN {X 0,Y 453.249,Z 434.962,A -85,B 0,C 180,E1 -8392.326,E2 -8392.326} C_VEL
LIN {X 0,Y 453.52,Z 427.171,A -85,B 0,C 180,E1 -8395.715,E2 -8395.715} C_VEL
LIN {X 0,Y 453.836,Z 419.372,A -85,B 0,C 180,E1 -8399.195,E2 -8399.195} C_VEL
LIN {X 0,Y 454.161,Z 412.707,A -85,B 0,C 180,E1 -8402.267,E2 -8402.267} C_VEL
LIN {X 0,Y 454.451,Z 406.026,A -85,B 0,C 180,E1 -8405.444,E2 -8405.444} C_VEL
LIN {X 0,Y 453.886,Z 401.291,A -85,B 0,C 180,E1 -8407.843,E2 -8407.843} C_VEL
LIN {X 0,Y 453.55,Z 398.992,A -85,B 0,C 180,E1 -8409.138,E2 -8409.138} C_VEL
LIN {X 0,Y 453.477,Z 398.997,A -85,B 0,C 180,E1 -8411.935,E2 -8411.935} C_VEL
LIN {X 0,Y 453.487,Z 398.995,A -85,B 0,C 180,E1 -8415.469,E2 -8415.469} C_VEL
LIN {X 0,Y 453.477,Z 398.996,A -85,B 0,C 180,E1 -8418.209,E2 -8418.209} C_VEL
LIN {X 0,Y 453.505,Z 398.998,A -85,B 0,C 180,E1 -8420.79,E2 -8420.79} C_VEL
LIN {X 0,Y 453.452,Z 399,A -85,B 0,C 180,E1 -8423.917,E2 -8423.917} C_VEL
LIN {X 0,Y 453.477,Z 398.997,A -85,B 0,C 180,E1 -8427.15,E2 -8427.15} C_VEL
LIN {X 0,Y 453.508,Z 398.995,A -85,B 0,C 180,E1 -8430.27,E2 -8430.27} C_VEL
LIN {X 0,Y 453.502,Z 398.994,A -85,B 0,C 180,E1 -8433.293,E2 -8433.293} C_VEL
LIN {X 0,Y 453.496,Z 398.997,A -85,B 0,C 180,E1 -8436.238,E2 -8436.238} C_VEL
LIN {X 0,Y 453.474,Z 398.997,A -85,B 0,C 180,E1 -8439.117,E2 -8439.117} C_VEL
LIN {X 0,Y 453.504,Z 398.995,A -85,B 0,C 180,E1 -8441.944,E2 -8441.944} C_VEL
LIN {X 0,Y 453.531,Z 398.99,A -85,B 0,C 180,E1 -8444.726,E2 -8444.726} C_VEL
LIN {X 0,Y 453.551,Z 398.989,A -85,B 0,C 180,E1 -8448.379,E2 -8448.379} C_VEL
LIN {X 0,Y 453.643,Z 398.979,A -85,B 0,C 180,E1 -8451.985,E2 -8451.985} C_VEL
LIN {X 0,Y 453.667,Z 398.974,A -85,B 0,C 180,E1 -8454.667,E2 -8454.667} C_VEL
LIN {X 0,Y 453.758,Z 398.963,A -85,B 0,C 180,E1 -8457.337,E2 -8457.337} C_VEL
LIN {X 0,Y 453.815,Z 398.956,A -85,B 0,C 180,E1 -8460,E2 -8460} C_VEL
LIN {X 0,Y 453.758,Z 398.964,A -85,B 0,C 180,E1 -8462.663,E2 -8462.663} C_VEL
LIN {X 0,Y 453.671,Z 398.973,A -85,B 0,C 180,E1 -8466.225,E2 -8466.225} C_VEL
LIN {X 0,Y 453.584,Z 398.985,A -85,B 0,C 180,E1 -8468.913,E2 -8468.913} C_VEL
LIN {X 0,Y 453.593,Z 398.986,A -85,B 0,C 180,E1 -8472.551,E2 -8472.551} C_VEL
LIN {X 0,Y 453.536,Z 398.991,A -85,B 0,C 180,E1 -8476.196,E2 -8476.196} C_VEL
LIN {X 0,Y 453.512,Z 398.993,A -85,B 0,C 180,E1 -8479.041,E2 -8479.041} C_VEL
LIN {X 0,Y 453.471,Z 398.998,A -85,B 0,C 180,E1 -8481.836,E2 -8481.836} C_VEL
LIN {X 0,Y 453.507,Z 398.993,A -85,B 0,C 180,E1 -8484.735,E2 -8484.735} C_VEL
LIN {X 0,Y 453.531,Z 398.993,A -85,B 0,C 180,E1 -8487.962,E2 -8487.962} C_VEL
LIN {X 0,Y 453.476,Z 398.997,A -85,B 0,C 180,E1 -8490.759,E2 -8490.759} C_VEL
LIN {X 0,Y 453.471,Z 399.002,A -85,B 0,C 180,E1 -8493.913,E2 -8493.913} C_VEL
LIN {X 0,Y 453.465,Z 398.997,A -85,B 0,C 180,E1 -8497.188,E2 -8497.188} C_VEL
LIN {X 0,Y 453.527,Z 398.991,A -85,B 0,C 180,E1 -8499.446,E2 -8499.446} C_VEL
LIN {X 0,Y 453.486,Z 398.994,A -85,B 0,C 180,E1 -8502.992,E2 -8502.992} C_VEL
LIN {X 0,Y 453.472,Z 399,A -85,B 0,C 180,E1 -8505.781,E2 -8505.781} C_VEL
LIN {X 0,Y 453.492,Z 398.993,A -85,B 0,C 180,E1 -8508.212,E2 -8508.212} C_VEL
LIN {X 0,Y 453.526,Z 398.988,A -85,B 0,C 180,E1 -8510.788,E2 -8510.788} C_VEL
LIN {X 0,Y 453.454,Z 398.998,A -85,B 0,C 180,E1 -8513.918,E2 -8513.918} C_VEL
LIN {X 0,Y 453.48,Z 398.999,A -85,B 0,C 180,E1 -8517.152,E2 -8517.152} C_VEL
LIN {X 0,Y 453.473,Z 398.995,A -85,B 0,C 180,E1 -8520.269,E2 -8520.269} C_VEL
LIN {X 0,Y 453.512,Z 398.995,A -85,B 0,C 180,E1 -8523.295,E2 -8523.295} C_VEL
LIN {X 0,Y 453.502,Z 398.992,A -85,B 0,C 180,E1 -8526.239,E2 -8526.239} C_VEL
LIN {X 0,Y 453.302,Z 399.023,A -85,B 0,C 180,E1 -8529.11,E2 -8529.11} C_VEL
LIN {X 0,Y 453.251,Z 402.853,A -85,B 0,C 180,E1 -8531.934,E2 -8531.934} C_VEL
LIN {X 0,Y 453.191,Z 406.776,A -85,B 0,C 180,E1 -8534.715,E2 -8534.715} C_VEL
LIN {X 0,Y 453.141,Z 411.089,A -85,B 0,C 180,E1 -8537.714,E2 -8537.714} C_VEL
LIN {X 0,Y 452.973,Z 416.03,A -85,B 0,C 180,E1 -8541.075,E2 -8541.075} C_VEL
LIN {X 0,Y 452.962,Z 418.616,A -85,B 0,C 180,E1 -8542.815,E2 -8542.815} C_VEL
LIN {X 0,Y 452.335,Z 419.762,A -85,B 0,C 180,E1 -8543.543,E2 -8543.543} C_VEL
LIN {X 0,Y 449.469,Z 421.776,A -85,B 0,C 180,E1 -8544.72,E2 -8544.72} C_VEL
LIN {X 0,Y 446.988,Z 423.403,A -85,B 0,C 180,E1 -8545.67,E2 -8545.67} C_VEL
LIN {X 0,Y 445.881,Z 424.591,A -85,B 0,C 180,E1 -8546.405,E2 -8546.405} C_VEL
LIN {X 0,Y 445.771,Z 424.973,A -85,B 0,C 180,E1 -8546.655,E2 -8546.655} C_VEL
LIN {X 0,Y 445.601,Z 426.999,A -85,B 0,C 180,E1 -8547.995,E2 -8547.995} C_VEL
LIN {X 0,Y 448.77,Z 442.381,A -85,B 0,C 180,E1 -8548.598,E2 -8548.598} C_VEL
LIN {X 0,Y 449.439,Z 447.122,A -85,B 0,C 180,E1 -8548.824,E2 -8548.824} C_VEL
LIN {X 0,Y 449.034,Z 458.96,A -85,B 0,C 180,E1 -8549.44,E2 -8549.44} C_VEL
LIN {X 0,Y 448.439,Z 470.448,A -85,B 0,C 180,E1 -8550.225,E2 -8550.225} C_VEL
LIN {X 0,Y 447.847,Z 482.009,A -85,B 0,C 180,E1 -8551.237,E2 -8551.237} C_VEL
LIN {X 0,Y 447.285,Z 491.361,A -85,B 0,C 180,E1 -8552.251,E2 -8552.251} C_VEL
LIN {X 0,Y 446.749,Z 499.91,A -85,B 0,C 180,E1 -8553.382,E2 -8553.382} C_VEL
LIN {X 0,Y 446.259,Z 508.217,A -85,B 0,C 180,E1 -8554.743,E2 -8554.743} C_VEL
LIN {X 0,Y 446.021,Z 514.902,A -85,B 0,C 180,E1 -8556.106,E2 -8556.106} C_VEL
LIN {X 0,Y 445.708,Z 521.067,A -85,B 0,C 180,E1 -8557.703,E2 -8557.703} C_VEL
LIN {X 0,Y 445.506,Z 525.078,A -85,B 0,C 180,E1 -8559.076,E2 -8559.076} C_VEL
LIN {X 0,Y 445.416,Z 527.142,A -85,B 0,C 180,E1 -8559.995,E2 -8559.995} C_VEL
LIN {X 0,Y 445.39,Z 528.782,A -85,B 0,C 180,E1 -8560.915,E2 -8560.915} C_VEL
LIN {X 0,Y 445.373,Z 530.129,A -85,B 0,C 180,E1 -8561.941,E2 -8561.941} C_VEL
LIN {X 0,Y 445.259,Z 531.183,A -85,B 0,C 180,E1 -8563.695,E2 -8563.695} C_VEL
LIN {X 0,Y 445.273,Z 531.159,A -85,B 0,C 180,E1 -8564.628,E2 -8564.628} C_VEL
LIN {X 0,Y 445.304,Z 530.614,A -85,B 0,C 180,E1 -8565.692,E2 -8565.692} C_VEL
LIN {X 0,Y 445.319,Z 528.497,A -85,B 0,C 180,E1 -8567.449,E2 -8567.449} C_VEL
LIN {X 0,Y 445.495,Z 525.764,A -85,B 0,C 180,E1 -8568.819,E2 -8568.819} C_VEL
LIN {X 0,Y 445.688,Z 521.675,A -85,B 0,C 180,E1 -8570.298,E2 -8570.298} C_VEL
LIN {X 0,Y 445.973,Z 515.956,A -85,B 0,C 180,E1 -8571.855,E2 -8571.855} C_VEL
LIN {X 0,Y 446.352,Z 509.724,A -85,B 0,C 180,E1 -8573.181,E2 -8573.181} C_VEL
LIN {X 0,Y 446.831,Z 501.197,A -85,B 0,C 180,E1 -8574.633,E2 -8574.633} C_VEL
LIN {X 0,Y 447.375,Z 492.374,A -85,B 0,C 180,E1 -8575.845,E2 -8575.845} C_VEL
LIN {X 0,Y 447.948,Z 483.126,A -85,B 0,C 180,E1 -8576.878,E2 -8576.878} C_VEL
LIN {X 0,Y 448.68,Z 471.683,A -85,B 0,C 180,E1 -8577.901,E2 -8577.901} C_VEL
LIN {X 0,Y 449.197,Z 460.661,A -85,B 0,C 180,E1 -8578.685,E2 -8578.685} C_VEL
LIN {X 0,Y 449.654,Z 449.985,A -85,B 0,C 180,E1 -8579.276,E2 -8579.276} C_VEL
LIN {X 0,Y 449.444,Z 444.839,A -85,B 0,C 180,E1 -8579.523,E2 -8579.523} C_VEL
LIN {X 0,Y 447.014,Z 433.062,A -85,B 0,C 180,E1 -8580.054,E2 -8580.054} C_VEL
LIN {X 0,Y 445.627,Z 427.176,A -85,B 0,C 180,E1 -8580.278,E2 -8580.278} C_VEL
LIN {X 0,Y 445.723,Z 422.47,A -85,B 0,C 180,E1 -8583.495,E2 -8583.495} C_VEL
LIN {X 0,Y 445.838,Z 417.741,A -85,B 0,C 180,E1 -8586.799,E2 -8586.799} C_VEL
LIN {X 0,Y 445.973,Z 414.03,A -85,B 0,C 180,E1 -8589.45,E2 -8589.45} C_VEL
LIN {X 0,Y 446.104,Z 409.679,A -85,B 0,C 180,E1 -8592.642,E2 -8592.642} C_VEL
LIN {X 0,Y 446.294,Z 405.057,A -85,B 0,C 180,E1 -8596.141,E2 -8596.141} C_VEL
LIN {X 0,Y 446.404,Z 401.281,A -85,B 0,C 180,E1 -8599.085,E2 -8599.085} C_VEL
LIN {X 0,Y 446.364,Z 399.888,A -85,B 0,C 180,E1 -8600.488,E2 -8600.488} C_VEL
LIN {X 0,Y 446.4,Z 399.885,A -85,B 0,C 180,E1 -8603.409,E2 -8603.409} C_VEL
LIN {X 0,Y 446.443,Z 399.88,A -85,B 0,C 180,E1 -8606.566,E2 -8606.566} C_VEL
LIN {X 0,Y 446.436,Z 399.877,A -85,B 0,C 180,E1 -8609.976,E2 -8609.976} C_VEL
LIN {X 0,Y 446.476,Z 399.873,A -85,B 0,C 180,E1 -8612.839,E2 -8612.839} C_VEL
LIN {X 0,Y 446.459,Z 399.874,A -85,B 0,C 180,E1 -8615.923,E2 -8615.923} C_VEL
LIN {X 0,Y 446.447,Z 399.877,A -85,B 0,C 180,E1 -8618.773,E2 -8618.773} C_VEL
LIN {X 0,Y 446.451,Z 399.877,A -85,B 0,C 180,E1 -8621.649,E2 -8621.649} C_VEL
LIN {X 0,Y 446.501,Z 399.869,A -85,B 0,C 180,E1 -8624.48,E2 -8624.48} C_VEL
LIN {X 0,Y 446.512,Z 399.864,A -85,B 0,C 180,E1 -8628.193,E2 -8628.193} C_VEL
LIN {X 0,Y 446.594,Z 399.857,A -85,B 0,C 180,E1 -8631.858,E2 -8631.858} C_VEL
LIN {X 0,Y 446.639,Z 399.85,A -85,B 0,C 180,E1 -8634.583,E2 -8634.583} C_VEL
LIN {X 0,Y 446.703,Z 399.841,A -85,B 0,C 180,E1 -8637.295,E2 -8637.295} C_VEL
LIN {X 0,Y 446.787,Z 399.832,A -85,B 0,C 180,E1 -8640,E2 -8640} C_VEL
LIN {X 0,Y 446.704,Z 399.844,A -85,B 0,C 180,E1 -8642.705,E2 -8642.705} C_VEL
LIN {X 0,Y 446.641,Z 399.849,A -85,B 0,C 180,E1 -8646.324,E2 -8646.324} C_VEL
LIN {X 0,Y 446.533,Z 399.863,A -85,B 0,C 180,E1 -8649.056,E2 -8649.056} C_VEL
LIN {X 0,Y 446.529,Z 399.865,A -85,B 0,C 180,E1 -8652.73,E2 -8652.73} C_VEL
LIN {X 0,Y 446.49,Z 399.869,A -85,B 0,C 180,E1 -8656.459,E2 -8656.459} C_VEL
LIN {X 0,Y 446.464,Z 399.874,A -85,B 0,C 180,E1 -8659.304,E2 -8659.304} C_VEL
LIN {X 0,Y 446.414,Z 399.881,A -85,B 0,C 180,E1 -8662.2,E2 -8662.2} C_VEL
LIN {X 0,Y 446.454,Z 399.876,A -85,B 0,C 180,E1 -8665.153,E2 -8665.153} C_VEL
LIN {X 0,Y 446.48,Z 399.872,A -85,B 0,C 180,E1 -8668.179,E2 -8668.179} C_VEL
LIN {X 0,Y 446.416,Z 399.879,A -85,B 0,C 180,E1 -8671.301,E2 -8671.301} C_VEL
LIN {X 0,Y 446.427,Z 399.876,A -85,B 0,C 180,E1 -8674.523,E2 -8674.523} C_VEL
LIN {X 0,Y 446.427,Z 399.873,A -85,B 0,C 180,E1 -8678.082,E2 -8678.082} C_VEL
LIN {X 0,Y 446.424,Z 399.877,A -85,B 0,C 180,E1 -8680.918,E2 -8680.918} C_VEL
LIN {X 0,Y 446.399,Z 399.881,A -85,B 0,C 180,E1 -8683.846,E2 -8683.846} C_VEL
LIN {X 0,Y 446.419,Z 399.878,A -85,B 0,C 180,E1 -8686.401,E2 -8686.401} C_VEL
LIN {X 0,Y 446.458,Z 399.947,A -85,B 0,C 180,E1 -8689.446,E2 -8689.446} C_VEL
LIN {X 0,Y 447.237,Z 404.584,A -85,B 0,C 180,E1 -8692.204,E2 -8692.204} C_VEL
LIN {X 0,Y 447.613,Z 408.682,A -85,B 0,C 180,E1 -8694.484,E2 -8694.484} C_VEL
LIN {X 0,Y 447.424,Z 412.857,A -85,B 0,C 180,E1 -8696.649,E2 -8696.649} C_VEL
LIN {X 0,Y 447.068,Z 419.257,A -85,B 0,C 180,E1 -8699.839,E2 -8699.839} C_VEL
LIN {X 0,Y 446.658,Z 425.56,A -85,B 0,C 180,E1 -8702.852,E2 -8702.852} C_VEL
LIN {X 0,Y 446.34,Z 432.295,A -85,B 0,C 180,E1 -8705.96,E2 -8705.96} C_VEL
LIN {X 0,Y 446.075,Z 439.599,A -85,B 0,C 180,E1 -8709.238,E2 -8709.238} C_VEL
LIN {X 0,Y 445.833,Z 447.205,A -85,B 0,C 180,E1 -8712.572,E2 -8712.572} C_VEL
LIN {X 0,Y 445.762,Z 449.952,A -85,B 0,C 180,E1 -8713.754,E2 -8713.754} C_VEL
LIN {X 0,Y 448.065,Z 463.199,A -85,B 0,C 180,E1 -8714.222,E2 -8714.222} C_VEL
LIN {X 0,Y 449.429,Z 474.582,A -85,B 0,C 180,E1 -8714.758,E2 -8714.758} C_VEL
LIN {X 0,Y 448.781,Z 487.582,A -85,B 0,C 180,E1 -8715.489,E2 -8715.489} C_VEL
LIN {X 0,Y 448.157,Z 498.381,A -85,B 0,C 180,E1 -8716.279,E2 -8716.279} C_VEL
LIN {X 0,Y 447.583,Z 509.424,A -85,B 0,C 180,E1 -8717.301,E2 -8717.301} C_VEL
LIN {X 0,Y 446.999,Z 519.283,A -85,B 0,C 180,E1 -8718.436,E2 -8718.436} C_VEL
LIN {X 0,Y 446.451,Z 527.379,A -85,B 0,C 180,E1 -8719.57,E2 -8719.57} C_VEL
LIN {X 0,Y 446.033,Z 535.339,A -85,B 0,C 180,E1 -8720.934,E2 -8720.934} C_VEL
LIN {X 0,Y 445.75,Z 541.715,A -85,B 0,C 180,E1 -8722.298,E2 -8722.298} C_VEL
LIN {X 0,Y 445.494,Z 547.636,A -85,B 0,C 180,E1 -8723.927,E2 -8723.927} C_VEL
LIN {X 0,Y 445.417,Z 551.815,A -85,B 0,C 180,E1 -8725.475,E2 -8725.475} C_VEL
LIN {X 0,Y 445.381,Z 553.66,A -85,B 0,C 180,E1 -8726.381,E2 -8726.381} C_VEL
LIN {X 0,Y 445.433,Z 555.047,A -85,B 0,C 180,E1 -8727.287,E2 -8727.287} C_VEL
LIN {X 0,Y 445.339,Z 556.636,A -85,B 0,C 180,E1 -8729.096,E2 -8729.096} C_VEL
LIN {X 0,Y 445.342,Z 556.838,A -85,B 0,C 180,E1 -8730,E2 -8730} C_VEL
LIN {X 0,Y 445.356,Z 555.994,A -85,B 0,C 180,E1 -8731.808,E2 -8731.808} C_VEL
LIN {X 0,Y 445.433,Z 554.991,A -85,B 0,C 180,E1 -8732.713,E2 -8732.713} C_VEL
LIN {X 0,Y 445.382,Z 553.574,A -85,B 0,C 180,E1 -8733.619,E2 -8733.619} C_VEL
LIN {X 0,Y 445.48,Z 550.617,A -85,B 0,C 180,E1 -8734.978,E2 -8734.978} C_VEL
LIN {X 0,Y 445.561,Z 545.162,A -85,B 0,C 180,E1 -8736.748,E2 -8736.748} C_VEL
LIN {X 0,Y 445.847,Z 539.428,A -85,B 0,C 180,E1 -8738.156,E2 -8738.156} C_VEL
LIN {X 0,Y 446.157,Z 532.467,A -85,B 0,C 180,E1 -8739.52,E2 -8739.52} C_VEL
LIN {X 0,Y 446.612,Z 523.733,A -85,B 0,C 180,E1 -8740.884,E2 -8740.884} C_VEL
LIN {X 0,Y 447.195,Z 514.784,A -85,B 0,C 180,E1 -8742.018,E2 -8742.018} C_VEL
LIN {X 0,Y 447.731,Z 503.988,A -85,B 0,C 180,E1 -8743.132,E2 -8743.132} C_VEL
LIN {X 0,Y 448.346,Z 492.525,A -85,B 0,C 180,E1 -8744.061,E2 -8744.061} C_VEL
LIN {X 0,Y 448.928,Z 479.954,A -85,B 0,C 180,E1 -8744.853,E2 -8744.853} C_VEL
LIN {X 0,Y 449.229,Z 473.152,A -85,B 0,C 180,E1 -8745.191,E2 -8745.191} C_VEL
LIN {X 0,Y 447.242,Z 459.334,A -85,B 0,C 180,E1 -8745.785,E2 -8745.785} C_VEL
LIN {X 0,Y 445.764,Z 450.122,A -85,B 0,C 180,E1 -8746.075,E2 -8746.075} C_VEL
LIN {X 0,Y 445.934,Z 442.505,A -85,B 0,C 180,E1 -8749.327,E2 -8749.327} C_VEL
LIN {X 0,Y 446.181,Z 435.841,A -85,B 0,C 180,E1 -8752.211,E2 -8752.211} C_VEL
LIN {X 0,Y 446.455,Z 428.067,A -85,B 0,C 180,E1 -8755.651,E2 -8755.651} C_VEL
LIN {X 0,Y 446.781,Z 420.27,A -85,B 0,C 180,E1 -8759.185,E2 -8759.185} C_VEL
LIN {X 0,Y 447.132,Z 413.603,A -85,B 0,C 180,E1 -8762.303,E2 -8762.303} C_VEL
LIN {X 0,Y 447.417,Z 406.925,A -85,B 0,C 180,E1 -8765.533,E2 -8765.533} C_VEL
LIN {X 0,Y 446.896,Z 402.458,A -85,B 0,C 180,E1 -8767.829,E2 -8767.829} C_VEL
LIN {X 0,Y 446.511,Z 399.869,A -85,B 0,C 180,E1 -8769.273,E2 -8769.273} C_VEL
LIN {X 0,Y 446.443,Z 399.877,A -85,B 0,C 180,E1 -8772.602,E2 -8772.602} C_VEL
LIN {X 0,Y 446.453,Z 399.875,A -85,B 0,C 180,E1 -8775.102,E2 -8775.102} C_VEL
LIN {X 0,Y 446.425,Z 399.877,A -85,B 0,C 180,E1 -8778.608,E2 -8778.608} C_VEL
LIN {X 0,Y 446.452,Z 399.874,A -85,B 0,C 180,E1 -8780.974,E2 -8780.974} C_VEL
LIN {X 0,Y 446.416,Z 399.878,A -85,B 0,C 180,E1 -8784.373,E2 -8784.373} C_VEL
LIN {X 0,Y 446.417,Z 399.876,A -85,B 0,C 180,E1 -8787.638,E2 -8787.638} C_VEL
LIN {X 0,Y 446.463,Z 399.872,A -85,B 0,C 180,E1 -8790.791,E2 -8790.791} C_VEL
LIN {X 0,Y 446.471,Z 399.87,A -85,B 0,C 180,E1 -8793.848,E2 -8793.848} C_VEL
LIN {X 0,Y 446.422,Z 399.876,A -85,B 0,C 180,E1 -8796.823,E2 -8796.823} C_VEL
LIN {X 0,Y 446.436,Z 399.875,A -85,B 0,C 180,E1 -8799.737,E2 -8799.737} C_VEL
LIN {X 0,Y 446.455,Z 399.872,A -85,B 0,C 180,E1 -8802.597,E2 -8802.597} C_VEL
LIN {X 0,Y 446.462,Z 399.872,A -85,B 0,C 180,E1 -8805.412,E2 -8805.412} C_VEL
LIN {X 0,Y 446.509,Z 399.867,A -85,B 0,C 180,E1 -8808.193,E2 -8808.193} C_VEL
LIN {X 0,Y 446.591,Z 399.857,A -85,B 0,C 180,E1 -8811.857,E2 -8811.857} C_VEL
LIN {X 0,Y 446.641,Z 399.849,A -85,B 0,C 180,E1 -8814.582,E2 -8814.582} C_VEL
LIN {X 0,Y 446.702,Z 399.842,A -85,B 0,C 180,E1 -8817.295,E2 -8817.295} C_VEL
LIN {X 0,Y 446.786,Z 399.831,A -85,B 0,C 180,E1 -8820,E2 -8820} C_VEL
LIN {X 0,Y 446.702,Z 399.843,A -85,B 0,C 180,E1 -8822.705,E2 -8822.705} C_VEL
LIN {X 0,Y 446.64,Z 399.85,A -85,B 0,C 180,E1 -8826.324,E2 -8826.324} C_VEL
LIN {X 0,Y 446.53,Z 399.863,A -85,B 0,C 180,E1 -8829.055,E2 -8829.055} C_VEL
LIN {X 0,Y 446.525,Z 399.865,A -85,B 0,C 180,E1 -8832.729,E2 -8832.729} C_VEL
LIN {X 0,Y 446.481,Z 399.872,A -85,B 0,C 180,E1 -8836.459,E2 -8836.459} C_VEL
LIN {X 0,Y 446.461,Z 399.871,A -85,B 0,C 180,E1 -8839.303,E2 -8839.303} C_VEL
LIN {X 0,Y 446.413,Z 399.88,A -85,B 0,C 180,E1 -8842.2,E2 -8842.2} C_VEL
LIN {X 0,Y 446.451,Z 399.872,A -85,B 0,C 180,E1 -8845.153,E2 -8845.153} C_VEL
LIN {X 0,Y 446.477,Z 399.872,A -85,B 0,C 180,E1 -8848.179,E2 -8848.179} C_VEL
LIN {X 0,Y 446.412,Z 399.876,A -85,B 0,C 180,E1 -8851.301,E2 -8851.301} C_VEL
LIN {X 0,Y 446.423,Z 399.875,A -85,B 0,C 180,E1 -8854.523,E2 -8854.523} C_VEL
LIN {X 0,Y 446.432,Z 399.876,A -85,B 0,C 180,E1 -8858.084,E2 -8858.084} C_VEL
LIN {X 0,Y 446.441,Z 399.871,A -85,B 0,C 180,E1 -8860.921,E2 -8860.921} C_VEL
LIN {X 0,Y 446.44,Z 399.876,A -85,B 0,C 180,E1 -8863.841,E2 -8863.841} C_VEL
LIN {X 0,Y 446.442,Z 399.871,A -85,B 0,C 180,E1 -8866.398,E2 -8866.398} C_VEL
LIN {X 0,Y 446.464,Z 399.871,A -85,B 0,C 180,E1 -8869.806,E2 -8869.806} C_VEL
LIN {X 0,Y 446.429,Z 399.872,A -85,B 0,C 180,E1 -8872.124,E2 -8872.124} C_VEL
LIN {X 0,Y 446.428,Z 399.878,A -85,B 0,C 180,E1 -8875.478,E2 -8875.478} C_VEL
LIN {X 0,Y 446.414,Z 399.875,A -85,B 0,C 180,E1 -8878.7,E2 -8878.7} C_VEL
LIN {X 0,Y 446.482,Z 399.867,A -85,B 0,C 180,E1 -8881.822,E2 -8881.822} C_VEL
LIN {X 0,Y 446.457,Z 399.873,A -85,B 0,C 180,E1 -8884.848,E2 -8884.848} C_VEL
LIN {X 0,Y 446.371,Z 399.881,A -85,B 0,C 180,E1 -8887.799,E2 -8887.799} C_VEL
LIN {X 0,Y 446.307,Z 399.892,A -85,B 0,C 180,E1 -8888.766,E2 -8888.766} C_VEL
LIN {X 0,Y 446.249,Z 400.631,A -85,B 0,C 180,E1 -8889.728,E2 -8889.728} C_VEL
LIN {X 0,Y 446.162,Z 404.565,A -85,B 0,C 180,E1 -8892.586,E2 -8892.586} C_VEL
LIN {X 0,Y 446.153,Z 407.201,A -85,B 0,C 180,E1 -8894.468,E2 -8894.468} C_VEL
LIN {X 0,Y 446.095,Z 411.685,A -85,B 0,C 180,E1 -8897.628,E2 -8897.628} C_VEL
LIN {X 0,Y 445.899,Z 416.483,A -85,B 0,C 180,E1 -8900.932,E2 -8900.932} C_VEL
LIN {X 0,Y 445.915,Z 420.493,A -85,B 0,C 180,E1 -8903.666,E2 -8903.666} C_VEL
LIN {X 0,Y 445.771,Z 424.973,A -85,B 0,C 180,E1 -8906.655,E2 -8906.655} C_VEL
LIN {X 0,Y 445.576,Z 426.387,A -85,B 0,C 180,E1 -8907.101,E2 -8907.101} C_VEL
LIN {X 0,Y 445.188,Z 428.788,A -85,B 0,C 180,E1 -8907.477,E2 -8907.477} C_VEL
LIN {X 0,Y 444.418,Z 433.504,A -85,B 0,C 180,E1 -8907.917,E2 -8907.917} C_VEL
LIN {X 0,Y 443.561,Z 439.167,A -85,B 0,C 180,E1 -8908.243,E2 -8908.243} C_VEL
LIN {X 0,Y 442.452,Z 451.284,A -85,B 0,C 180,E1 -8908.796,E2 -8908.796} C_VEL
LIN {X 0,Y 441.901,Z 464.043,A -85,B 0,C 180,E1 -8909.545,E2 -8909.545} C_VEL
LIN {X 0,Y 441.32,Z 474.532,A -85,B 0,C 180,E1 -8910.342,E2 -8910.342} C_VEL
LIN {X 0,Y 440.666,Z 485.284,A -85,B 0,C 180,E1 -8911.371,E2 -8911.371} C_VEL
LIN {X 0,Y 440.087,Z 494.956,A -85,B 0,C 180,E1 -8912.517,E2 -8912.517} C_VEL
LIN {X 0,Y 439.557,Z 502.908,A -85,B 0,C 180,E1 -8913.667,E2 -8913.667} C_VEL
LIN {X 0,Y 439.13,Z 510.701,A -85,B 0,C 180,E1 -8915.05,E2 -8915.05} C_VEL
LIN {X 0,Y 438.877,Z 516.928,A -85,B 0,C 180,E1 -8916.436,E2 -8916.436} C_VEL
LIN {X 0,Y 438.609,Z 521.905,A -85,B 0,C 180,E1 -8917.828,E2 -8917.828} C_VEL
LIN {X 0,Y 438.423,Z 525.757,A -85,B 0,C 180,E1 -8919.224,E2 -8919.224} C_VEL
LIN {X 0,Y 438.328,Z 527.744,A -85,B 0,C 180,E1 -8920.158,E2 -8920.158} C_VEL
LIN {X 0,Y 438.289,Z 529.312,A -85,B 0,C 180,E1 -8921.094,E2 -8921.094} C_VEL
LIN {X 0,Y 438.277,Z 530.423,A -85,B 0,C 180,E1 -8922.032,E2 -8922.032} C_VEL
LIN {X 0,Y 438.195,Z 531.123,A -85,B 0,C 180,E1 -8922.976,E2 -8922.976} C_VEL
LIN {X 0,Y 438.157,Z 531.425,A -85,B 0,C 180,E1 -8923.922,E2 -8923.922} C_VEL
LIN {X 0,Y 438.188,Z 531.317,A -85,B 0,C 180,E1 -8924.869,E2 -8924.869} C_VEL
LIN {X 0,Y 438.2,Z 530.749,A -85,B 0,C 180,E1 -8925.822,E2 -8925.822} C_VEL
LIN {X 0,Y 438.198,Z 529.769,A -85,B 0,C 180,E1 -8926.779,E2 -8926.779} C_VEL
LIN {X 0,Y 438.26,Z 528.37,A -85,B 0,C 180,E1 -8927.739,E2 -8927.739} C_VEL
LIN {X 0,Y 438.441,Z 525.874,A -85,B 0,C 180,E1 -8928.961,E2 -8928.961} C_VEL
LIN {X 0,Y 438.674,Z 521.21,A -85,B 0,C 180,E1 -8930.638,E2 -8930.638} C_VEL
LIN {X 0,Y 439.057,Z 514.639,A -85,B 0,C 180,E1 -8932.355,E2 -8932.355} C_VEL
LIN {X 0,Y 439.5,Z 507.644,A -85,B 0,C 180,E1 -8933.782,E2 -8933.782} C_VEL
LIN {X 0,Y 440.01,Z 499.998,A -85,B 0,C 180,E1 -8935.041,E2 -8935.041} C_VEL
LIN {X 0,Y 440.622,Z 489.738,A -85,B 0,C 180,E1 -8936.398,E2 -8936.398} C_VEL
LIN {X 0,Y 441.348,Z 479.306,A -85,B 0,C 180,E1 -8937.503,E2 -8937.503} C_VEL
LIN {X 0,Y 442.041,Z 467.49,A -85,B 0,C 180,E1 -8938.487,E2 -8938.487} C_VEL
LIN {X 0,Y 442.671,Z 454.907,A -85,B 0,C 180,E1 -8939.298,E2 -8939.298} C_VEL
LIN {X 0,Y 442.896,Z 447.543,A -85,B 0,C 180,E1 -8939.67,E2 -8939.67} C_VEL
LIN {X 0,Y 440.556,Z 435.687,A -85,B 0,C 180,E1 -8940.245,E2 -8940.245} C_VEL
LIN {X 0,Y 438.549,Z 427.367,A -85,B 0,C 180,E1 -8940.586,E2 -8940.586} C_VEL
LIN {X 0,Y 438.663,Z 422.303,A -85,B 0,C 180,E1 -8944.107,E2 -8944.107} C_VEL
LIN {X 0,Y 438.818,Z 417.55,A -85,B 0,C 180,E1 -8947.488,E2 -8947.488} C_VEL
LIN {X 0,Y 438.939,Z 414.353,A -85,B 0,C 180,E1 -8949.825,E2 -8949.825} C_VEL
LIN {X 0,Y 439.125,Z 409.448,A -85,B 0,C 180,E1 -8953.487,E2 -8953.487} C_VEL
LIN {X 0,Y 439.286,Z 405.503,A -85,B 0,C 180,E1 -8956.533,E2 -8956.533} C_VEL
LIN {X 0,Y 439.372,Z 402.383,A -85,B 0,C 180,E1 -8959.018,E2 -8959.018} C_VEL
LIN {X 0,Y 439.316,Z 400.927,A -85,B 0,C 180,E1 -8960.215,E2 -8960.215} C_VEL
LIN {X 0,Y 439.346,Z 400.763,A -85,B 0,C 180,E1 -8963.112,E2 -8963.112} C_VEL
LIN {X 0,Y 439.391,Z 400.757,A -85,B 0,C 180,E1 -8966.276,E2 -8966.276} C_VEL
LIN {X 0,Y 439.409,Z 400.754,A -85,B 0,C 180,E1 -8969.732,E2 -8969.732} C_VEL
LIN {X 0,Y 439.439,Z 400.748,A -85,B 0,C 180,E1 -8972.368,E2 -8972.368} C_VEL
LIN {X 0,Y 439.409,Z 400.752,A -85,B 0,C 180,E1 -8975.735,E2 -8975.735} C_VEL
LIN {X 0,Y 439.382,Z 400.754,A -85,B 0,C 180,E1 -8979.397,E2 -8979.397} C_VEL
LIN {X 0,Y 439.425,Z 400.747,A -85,B 0,C 180,E1 -8982.309,E2 -8982.309} C_VEL
LIN {X 0,Y 439.441,Z 400.745,A -85,B 0,C 180,E1 -8985.174,E2 -8985.174} C_VEL
LIN {X 0,Y 439.478,Z 400.742,A -85,B 0,C 180,E1 -8988.001,E2 -8988.001} C_VEL
LIN {X 0,Y 439.542,Z 400.734,A -85,B 0,C 180,E1 -8991.726,E2 -8991.726} C_VEL
LIN {X 0,Y 439.615,Z 400.725,A -85,B 0,C 180,E1 -8994.496,E2 -8994.496} C_VEL
LIN {X 0,Y 439.63,Z 400.725,A -85,B 0,C 180,E1 -8998.168,E2 -8998.168} C_VEL
LIN {X 0,Y 439.757,Z 400.707,A -85,B 0,C 180,E1 -9000,E2 -9000} C_VEL
LIN {X 0,Y 439.651,Z 400.722,A -85,B 0,C 180,E1 -9002.749,E2 -9002.749} C_VEL
LIN {X 0,Y 439.612,Z 400.724,A -85,B 0,C 180,E1 -9006.425,E2 -9006.425} C_VEL
LIN {X 0,Y 439.495,Z 400.739,A -85,B 0,C 180,E1 -9009.202,E2 -9009.202} C_VEL
LIN {X 0,Y 439.499,Z 400.74,A -85,B 0,C 180,E1 -9012.727,E2 -9012.727} C_VEL
LIN {X 0,Y 439.455,Z 400.746,A -85,B 0,C 180,E1 -9016.355,E2 -9016.355} C_VEL
LIN {X 0,Y 439.397,Z 400.753,A -85,B 0,C 180,E1 -9019.627,E2 -9019.627} C_VEL
LIN {X 0,Y 439.36,Z 400.758,A -85,B 0,C 180,E1 -9022.576,E2 -9022.576} C_VEL
LIN {X 0,Y 439.401,Z 400.752,A -85,B 0,C 180,E1 -9025.585,E2 -9025.585} C_VEL
LIN {X 0,Y 439.421,Z 400.749,A -85,B 0,C 180,E1 -9028.673,E2 -9028.673} C_VEL
LIN {X 0,Y 439.371,Z 400.755,A -85,B 0,C 180,E1 -9031.861,E2 -9031.861} C_VEL
LIN {X 0,Y 439.397,Z 400.753,A -85,B 0,C 180,E1 -9035.156,E2 -9035.156} C_VEL
LIN {X 0,Y 439.381,Z 400.753,A -85,B 0,C 180,E1 -9038.595,E2 -9038.595} C_VEL
LIN {X 0,Y 439.386,Z 400.755,A -85,B 0,C 180,E1 -9041.257,E2 -9041.257} C_VEL
LIN {X 0,Y 439.4,Z 400.754,A -85,B 0,C 180,E1 -9044.73,E2 -9044.73} C_VEL
LIN {X 0,Y 439.396,Z 400.754,A -85,B 0,C 180,E1 -9047.797,E2 -9047.797} C_VEL
LIN {X 0,Y 439.414,Z 400.889,A -85,B 0,C 180,E1 -9049.168,E2 -9049.168} C_VEL
LIN {X 0,Y 440.077,Z 404.708,A -85,B 0,C 180,E1 -9051.493,E2 -9051.493} C_VEL
LIN {X 0,Y 440.609,Z 408.714,A -85,B 0,C 180,E1 -9053.831,E2 -9053.831} C_VEL
LIN {X 0,Y 440.56,Z 412.876,A -85,B 0,C 180,E1 -9056.06,E2 -9056.06} C_VEL
LIN {X 0,Y 440.064,Z 419.808,A -85,B 0,C 180,E1 -9059.588,E2 -9059.588} C_VEL
LIN {X 0,Y 439.662,Z 425.531,A -85,B 0,C 180,E1 -9062.383,E2 -9062.383} C_VEL
LIN {X 0,Y 439.31,Z 432.683,A -85,B 0,C 180,E1 -9065.766,E2 -9065.766} C_VEL
LIN {X 0,Y 439.062,Z 439.505,A -85,B 0,C 180,E1 -9068.891,E2 -9068.891} C_VEL
LIN {X 0,Y 438.76,Z 447.088,A -85,B 0,C 180,E1 -9072.282,E2 -9072.282} C_VEL
LIN {X 0,Y 438.728,Z 449.729,A -85,B 0,C 180,E1 -9073.45,E2 -9073.45} C_VEL
LIN {X 0,Y 441.182,Z 463.538,A -85,B 0,C 180,E1 -9073.962,E2 -9073.962} C_VEL
LIN {X 0,Y 442.592,Z 474.854,A -85,B 0,C 180,E1 -9074.516,E2 -9074.516} C_VEL
LIN {X 0,Y 441.918,Z 487.731,A -85,B 0,C 180,E1 -9075.259,E2 -9075.259} C_VEL
LIN {X 0,Y 441.265,Z 498.448,A -85,B 0,C 180,E1 -9076.061,E2 -9076.061} C_VEL
LIN {X 0,Y 440.659,Z 509.423,A -85,B 0,C 180,E1 -9077.098,E2 -9077.098} C_VEL
LIN {X 0,Y 440.034,Z 519.247,A -85,B 0,C 180,E1 -9078.25,E2 -9078.25} C_VEL
LIN {X 0,Y 439.446,Z 527.315,A -85,B 0,C 180,E1 -9079.402,E2 -9079.402} C_VEL
LIN {X 0,Y 438.997,Z 535.247,A -85,B 0,C 180,E1 -9080.788,E2 -9080.788} C_VEL
LIN {X 0,Y 438.703,Z 541.595,A -85,B 0,C 180,E1 -9082.174,E2 -9082.174} C_VEL
LIN {X 0,Y 438.446,Z 546.875,A -85,B 0,C 180,E1 -9083.629,E2 -9083.629} C_VEL
LIN {X 0,Y 438.346,Z 551.654,A -85,B 0,C 180,E1 -9085.402,E2 -9085.402} C_VEL
LIN {X 0,Y 438.282,Z 553.485,A -85,B 0,C 180,E1 -9086.322,E2 -9086.322} C_VEL
LIN {X 0,Y 438.341,Z 554.864,A -85,B 0,C 180,E1 -9087.243,E2 -9087.243} C_VEL
LIN {X 0,Y 438.252,Z 556.44,A -85,B 0,C 180,E1 -9089.081,E2 -9089.081} C_VEL
LIN {X 0,Y 438.253,Z 556.632,A -85,B 0,C 180,E1 -9090,E2 -9090} C_VEL
LIN {X 0,Y 438.278,Z 555.775,A -85,B 0,C 180,E1 -9091.838,E2 -9091.838} C_VEL
LIN {X 0,Y 438.341,Z 554.766,A -85,B 0,C 180,E1 -9092.757,E2 -9092.757} C_VEL
LIN {X 0,Y 438.283,Z 553.337,A -85,B 0,C 180,E1 -9093.677,E2 -9093.677} C_VEL
LIN {X 0,Y 438.39,Z 550.367,A -85,B 0,C 180,E1 -9095.058,E2 -9095.058} C_VEL
LIN {X 0,Y 438.448,Z 546.342,A -85,B 0,C 180,E1 -9096.442,E2 -9096.442} C_VEL
LIN {X 0,Y 438.722,Z 540.145,A -85,B 0,C 180,E1 -9098.057,E2 -9098.057} C_VEL
LIN {X 0,Y 439.063,Z 533.387,A -85,B 0,C 180,E1 -9099.443,E2 -9099.443} C_VEL
LIN {X 0,Y 439.492,Z 524.993,A -85,B 0,C 180,E1 -9100.83,E2 -9100.83} C_VEL
LIN {X 0,Y 440.081,Z 516.346,A -85,B 0,C 180,E1 -9101.982,E2 -9101.982} C_VEL
LIN {X 0,Y 440.649,Z 506.312,A -85,B 0,C 180,E1 -9103.074,E2 -9103.074} C_VEL
LIN {X 0,Y 441.275,Z 495.098,A -85,B 0,C 180,E1 -9104.056,E2 -9104.056} C_VEL
LIN {X 0,Y 441.853,Z 483.343,A -85,B 0,C 180,E1 -9104.861,E2 -9104.861} C_VEL
LIN {X 0,Y 442.25,Z 473.708,A -85,B 0,C 180,E1 -9105.378,E2 -9105.378} C_VEL
LIN {X 0,Y 440.368,Z 460.291,A -85,B 0,C 180,E1 -9105.976,E2 -9105.976} C_VEL
LIN {X 0,Y 438.717,Z 449.855,A -85,B 0,C 180,E1 -9106.341,E2 -9106.341} C_VEL
LIN {X 0,Y 438.867,Z 442.25,A -85,B 0,C 180,E1 -9109.651,E2 -9109.651} C_VEL
LIN {X 0,Y 439.109,Z 435.613,A -85,B 0,C 180,E1 -9112.589,E2 -9112.589} C_VEL
LIN {X 0,Y 439.379,Z 428.934,A -85,B 0,C 180,E1 -9115.586,E2 -9115.586} C_VEL
LIN {X 0,Y 439.736,Z 421.169,A -85,B 0,C 180,E1 -9119.173,E2 -9119.173} C_VEL
LIN {X 0,Y 440.082,Z 414.83,A -85,B 0,C 180,E1 -9122.178,E2 -9122.178} C_VEL
LIN {X 0,Y 440.392,Z 408.007,A -85,B 0,C 180,E1 -9125.522,E2 -9125.522} C_VEL
LIN {X 0,Y 439.866,Z 403.455,A -85,B 0,C 180,E1 -9127.906,E2 -9127.906} C_VEL
LIN {X 0,Y 439.461,Z 400.746,A -85,B 0,C 180,E1 -9129.47,E2 -9129.47} C_VEL
LIN {X 0,Y 439.396,Z 400.754,A -85,B 0,C 180,E1 -9132.629,E2 -9132.629} C_VEL
LIN {X 0,Y 439.403,Z 400.751,A -85,B 0,C 180,E1 -9135.271,E2 -9135.271} C_VEL
LIN {X 0,Y 439.385,Z 400.755,A -85,B 0,C 180,E1 -9138.742,E2 -9138.742} C_VEL
LIN {X 0,Y 439.38,Z 400.752,A -85,B 0,C 180,E1 -9141.605,E2 -9141.605} C_VEL
LIN {X 0,Y 439.395,Z 400.754,A -85,B 0,C 180,E1 -9144.843,E2 -9144.843} C_VEL
LIN {X 0,Y 439.369,Z 400.755,A -85,B 0,C 180,E1 -9148.139,E2 -9148.139} C_VEL
LIN {X 0,Y 439.419,Z 400.748,A -85,B 0,C 180,E1 -9151.326,E2 -9151.326} C_VEL
LIN {X 0,Y 439.398,Z 400.754,A -85,B 0,C 180,E1 -9154.414,E2 -9154.414} C_VEL
LIN {X 0,Y 439.358,Z 400.757,A -85,B 0,C 180,E1 -9157.424,E2 -9157.424} C_VEL
LIN {X 0,Y 439.433,Z 400.747,A -85,B 0,C 180,E1 -9160.662,E2 -9160.662} C_VEL
LIN {X 0,Y 439.454,Z 400.747,A -85,B 0,C 180,E1 -9164.224,E2 -9164.224} C_VEL
LIN {X 0,Y 439.475,Z 400.743,A -85,B 0,C 180,E1 -9168.001,E2 -9168.001} C_VEL
LIN {X 0,Y 439.539,Z 400.734,A -85,B 0,C 180,E1 -9171.726,E2 -9171.726} C_VEL
LIN {X 0,Y 439.616,Z 400.724,A -85,B 0,C 180,E1 -9174.496,E2 -9174.496} C_VEL
LIN {X 0,Y 439.627,Z 400.723,A -85,B 0,C 180,E1 -9178.168,E2 -9178.168} C_VEL
LIN {X 0,Y 439.756,Z 400.707,A -85,B 0,C 180,E1 -9180,E2 -9180} C_VEL
LIN {X 0,Y 439.649,Z 400.722,A -85,B 0,C 180,E1 -9182.749,E2 -9182.749} C_VEL
LIN {X 0,Y 439.611,Z 400.726,A -85,B 0,C 180,E1 -9186.425,E2 -9186.425} C_VEL
LIN {X 0,Y 439.492,Z 400.739,A -85,B 0,C 180,E1 -9189.202,E2 -9189.202} C_VEL
LIN {X 0,Y 439.465,Z 400.743,A -85,B 0,C 180,E1 -9192.937,E2 -9192.937} C_VEL
LIN {X 0,Y 439.438,Z 400.749,A -85,B 0,C 180,E1 -9196.349,E2 -9196.349} C_VEL
LIN {X 0,Y 439.395,Z 400.751,A -85,B 0,C 180,E1 -9199.626,E2 -9199.626} C_VEL
LIN {X 0,Y 439.359,Z 400.756,A -85,B 0,C 180,E1 -9202.576,E2 -9202.576} C_VEL
LIN {X 0,Y 439.398,Z 400.751,A -85,B 0,C 180,E1 -9205.585,E2 -9205.585} C_VEL
LIN {X 0,Y 439.417,Z 400.748,A -85,B 0,C 180,E1 -9208.673,E2 -9208.673} C_VEL
LIN {X 0,Y 439.375,Z 400.757,A -85,B 0,C 180,E1 -9212.034,E2 -9212.034} C_VEL
LIN {X 0,Y 439.389,Z 400.751,A -85,B 0,C 180,E1 -9215.341,E2 -9215.341} C_VEL
LIN {X 0,Y 439.393,Z 400.75,A -85,B 0,C 180,E1 -9218.594,E2 -9218.594} C_VEL
LIN {X 0,Y 439.399,Z 400.75,A -85,B 0,C 180,E1 -9221.26,E2 -9221.26} C_VEL
LIN {X 0,Y 439.405,Z 400.748,A -85,B 0,C 180,E1 -9224.729,E2 -9224.729} C_VEL
LIN {X 0,Y 439.408,Z 400.751,A -85,B 0,C 180,E1 -9227.798,E2 -9227.798} C_VEL
LIN {X 0,Y 439.446,Z 400.742,A -85,B 0,C 180,E1 -9230.231,E2 -9230.231} C_VEL
LIN {X 0,Y 439.374,Z 400.754,A -85,B 0,C 180,E1 -9233.714,E2 -9233.714} C_VEL
LIN {X 0,Y 439.37,Z 400.755,A -85,B 0,C 180,E1 -9237.055,E2 -9237.055} C_VEL
LIN {X 0,Y 439.38,Z 400.751,A -85,B 0,C 180,E1 -9240.275,E2 -9240.275} C_VEL
LIN {X 0,Y 439.428,Z 400.748,A -85,B 0,C 180,E1 -9243.397,E2 -9243.397} C_VEL
LIN {X 0,Y 439.382,Z 400.752,A -85,B 0,C 180,E1 -9246.43,E2 -9246.43} C_VEL
LIN {X 0,Y 439.328,Z 400.758,A -85,B 0,C 180,E1 -9248.412,E2 -9248.412} C_VEL
LIN {X 0,Y 439.2,Z 401.024,A -85,B 0,C 180,E1 -9249.389,E2 -9249.389} C_VEL
LIN {X 0,Y 439.125,Z 404.974,A -85,B 0,C 180,E1 -9252.297,E2 -9252.297} C_VEL
LIN {X 0,Y 439.016,Z 408.929,A -85,B 0,C 180,E1 -9255.16,E2 -9255.16} C_VEL
LIN {X 0,Y 438.989,Z 412.919,A -85,B 0,C 180,E1 -9257.988,E2 -9257.988} C_VEL
LIN {X 0,Y 438.828,Z 418.272,A -85,B 0,C 180,E1 -9261.713,E2 -9261.713} C_VEL
LIN {X 0,Y 438.848,Z 420.968,A -85,B 0,C 180,E1 -9263.564,E2 -9263.564} C_VEL
LIN {X 0,Y 438.741,Z 425.039,A -85,B 0,C 180,E1 -9266.327,E2 -9266.327} C_VEL
LIN {X 0,Y 438.57,Z 427.186,A -85,B 0,C 180,E1 -9267.762,E2 -9267.762} C_VEL
LIN {X 0,Y 441.527,Z 441.8,A -85,B 0,C 180,E1 -9268.333,E2 -9268.333} C_VEL
LIN {X 0,Y 442.546,Z 447.994,A -85,B 0,C 180,E1 -9268.635,E2 -9268.635} C_VEL
LIN {X 0,Y 442.452,Z 451.284,A -85,B 0,C 180,E1 -9268.796,E2 -9268.796} C_VEL
LIN {X 0,Y 441.647,Z 456.82,A -85,B 0,C 180,E1 -9269.073,E2 -9269.073} C_VEL
LIN {X 0,Y 438.398,Z 465.508,A -85,B 0,C 180,E1 -9269.537,E2 -9269.537} C_VEL
LIN {X 0,Y 435.084,Z 473.798,A -85,B 0,C 180,E1 -9270.089,E2 -9270.089} C_VEL
LIN {X 0,Y 434.164,Z 478.66,A -85,B 0,C 180,E1 -9270.503,E2 -9270.503} C_VEL
LIN {X 0,Y 433.46,Z 489.347,A -85,B 0,C 180,E1 -9271.626,E2 -9271.626} C_VEL
LIN {X 0,Y 432.867,Z 498.309,A -85,B 0,C 180,E1 -9272.792,E2 -9272.792} C_VEL
LIN {X 0,Y 432.304,Z 507.069,A -85,B 0,C 180,E1 -9274.195,E2 -9274.195} C_VEL
LIN {X 0,Y 431.881,Z 514.079,A -85,B 0,C 180,E1 -9275.603,E2 -9275.603} C_VEL
LIN {X 0,Y 431.692,Z 519.509,A -85,B 0,C 180,E1 -9276.966,E2 -9276.966} C_VEL
LIN {X 0,Y 431.413,Z 524.097,A -85,B 0,C 180,E1 -9278.431,E2 -9278.431} C_VEL
LIN {X 0,Y 431.324,Z 526.435,A -85,B 0,C 180,E1 -9279.378,E2 -9279.378} C_VEL
LIN {X 0,Y 431.246,Z 528.346,A -85,B 0,C 180,E1 -9280.327,E2 -9280.327} C_VEL
LIN {X 0,Y 431.177,Z 530.649,A -85,B 0,C 180,E1 -9282.048,E2 -9282.048} C_VEL
LIN {X 0,Y 431.085,Z 531.437,A -85,B 0,C 180,E1 -9283.194,E2 -9283.194} C_VEL
LIN {X 0,Y 431.059,Z 531.655,A -85,B 0,C 180,E1 -9284.156,E2 -9284.156} C_VEL
LIN {X 0,Y 431.102,Z 530.95,A -85,B 0,C 180,E1 -9285.879,E2 -9285.879} C_VEL
LIN {X 0,Y 431.134,Z 529.719,A -85,B 0,C 180,E1 -9287.063,E2 -9287.063} C_VEL
LIN {X 0,Y 431.284,Z 527.262,A -85,B 0,C 180,E1 -9288.527,E2 -9288.527} C_VEL
LIN {X 0,Y 431.512,Z 523.725,A -85,B 0,C 180,E1 -9290,E2 -9290} C_VEL
LIN {X 0,Y 431.792,Z 519.035,A -85,B 0,C 180,E1 -9291.466,E2 -9291.466} C_VEL
LIN {X 0,Y 432.167,Z 512.819,A -85,B 0,C 180,E1 -9292.972,E2 -9292.972} C_VEL
LIN {X 0,Y 432.61,Z 506.179,A -85,B 0,C 180,E1 -9294.268,E2 -9294.268} C_VEL
LIN {X 0,Y 433.268,Z 497.001,A -85,B 0,C 180,E1 -9295.716,E2 -9295.716} C_VEL
LIN {X 0,Y 433.905,Z 487.023,A -85,B 0,C 180,E1 -9296.969,E2 -9296.969} C_VEL
LIN {X 0,Y 434.71,Z 475.807,A -85,B 0,C 180,E1 -9298.09,E2 -9298.09} C_VEL
LIN {X 0,Y 435.376,Z 464.792,A -85,B 0,C 180,E1 -9298.964,E2 -9298.964} C_VEL
LIN {X 0,Y 436.018,Z 452.403,A -85,B 0,C 180,E1 -9299.716,E2 -9299.716} C_VEL
LIN {X 0,Y 436.053,Z 448.279,A -85,B 0,C 180,E1 -9299.929,E2 -9299.929} C_VEL
LIN {X 0,Y 433.545,Z 435.809,A -85,B 0,C 180,E1 -9300.55,E2 -9300.55} C_VEL
LIN {X 0,Y 431.498,Z 427.561,A -85,B 0,C 180,E1 -9300.912,E2 -9300.912} C_VEL
LIN {X 0,Y 431.601,Z 423.385,A -85,B 0,C 180,E1 -9303.854,E2 -9303.854} C_VEL
LIN {X 0,Y 431.756,Z 418.888,A -85,B 0,C 180,E1 -9307.098,E2 -9307.098} C_VEL
LIN {X 0,Y 431.884,Z 414.814,A -85,B 0,C 180,E1 -9310.109,E2 -9310.109} C_VEL
LIN {X 0,Y 432.07,Z 410.874,A -85,B 0,C 180,E1 -9313.091,E2 -9313.091} C_VEL
LIN {X 0,Y 432.287,Z 405.984,A -85,B 0,C 180,E1 -9316.935,E2 -9316.935} C_VEL
LIN {X 0,Y 432.319,Z 402.433,A -85,B 0,C 180,E1 -9319.822,E2 -9319.822} C_VEL
LIN {X 0,Y 432.274,Z 401.643,A -85,B 0,C 180,E1 -9320.649,E2 -9320.649} C_VEL
LIN {X 0,Y 432.306,Z 401.64,A -85,B 0,C 180,E1 -9323.022,E2 -9323.022} C_VEL
LIN {X 0,Y 432.355,Z 401.633,A -85,B 0,C 180,E1 -9325.996,E2 -9325.996} C_VEL
LIN {X 0,Y 432.39,Z 401.628,A -85,B 0,C 180,E1 -9329.744,E2 -9329.744} C_VEL
LIN {X 0,Y 432.395,Z 401.624,A -85,B 0,C 180,E1 -9333.372,E2 -9333.372} C_VEL
LIN {X 0,Y 432.365,Z 401.628,A -85,B 0,C 180,E1 -9336.023,E2 -9336.023} C_VEL
LIN {X 0,Y 432.344,Z 401.631,A -85,B 0,C 180,E1 -9339.046,E2 -9339.046} C_VEL
LIN {X 0,Y 432.372,Z 401.627,A -85,B 0,C 180,E1 -9342.011,E2 -9342.011} C_VEL
LIN {X 0,Y 432.389,Z 401.625,A -85,B 0,C 180,E1 -9344.926,E2 -9344.926} C_VEL
LIN {X 0,Y 432.453,Z 401.618,A -85,B 0,C 180,E1 -9347.803,E2 -9347.803} C_VEL
LIN {X 0,Y 432.486,Z 401.613,A -85,B 0,C 180,E1 -9351.59,E2 -9351.59} C_VEL
LIN {X 0,Y 432.591,Z 401.599,A -85,B 0,C 180,E1 -9354.406,E2 -9354.406} C_VEL
LIN {X 0,Y 432.6,Z 401.601,A -85,B 0,C 180,E1 -9358.138,E2 -9358.138} C_VEL
LIN {X 0,Y 432.727,Z 401.583,A -85,B 0,C 180,E1 -9360,E2 -9360} C_VEL
LIN {X 0,Y 432.6,Z 401.6,A -85,B 0,C 180,E1 -9362.794,E2 -9362.794} C_VEL
LIN {X 0,Y 432.567,Z 401.602,A -85,B 0,C 180,E1 -9366.531,E2 -9366.531} C_VEL
LIN {X 0,Y 432.439,Z 401.618,A -85,B 0,C 180,E1 -9369.353,E2 -9369.353} C_VEL
LIN {X 0,Y 432.44,Z 401.62,A -85,B 0,C 180,E1 -9372.812,E2 -9372.812} C_VEL
LIN {X 0,Y 432.417,Z 401.622,A -85,B 0,C 180,E1 -9376.484,E2 -9376.484} C_VEL
LIN {X 0,Y 432.334,Z 401.633,A -85,B 0,C 180,E1 -9379.961,E2 -9379.961} C_VEL
LIN {X 0,Y 432.315,Z 401.636,A -85,B 0,C 180,E1 -9382.965,E2 -9382.965} C_VEL
LIN {X 0,Y 432.36,Z 401.63,A -85,B 0,C 180,E1 -9386.033,E2 -9386.033} C_VEL
LIN {X 0,Y 432.348,Z 401.632,A -85,B 0,C 180,E1 -9389.187,E2 -9389.187} C_VEL
LIN {X 0,Y 432.322,Z 401.636,A -85,B 0,C 180,E1 -9392.294,E2 -9392.294} C_VEL
LIN {X 0,Y 432.337,Z 401.631,A -85,B 0,C 180,E1 -9394.678,E2 -9394.678} C_VEL
LIN {X 0,Y 432.342,Z 401.627,A -85,B 0,C 180,E1 -9398.15,E2 -9398.15} C_VEL
LIN {X 0,Y 432.33,Z 401.635,A -85,B 0,C 180,E1 -9401.603,E2 -9401.603} C_VEL
LIN {X 0,Y 432.332,Z 401.634,A -85,B 0,C 180,E1 -9404.348,E2 -9404.348} C_VEL
LIN {X 0,Y 432.323,Z 401.635,A -85,B 0,C 180,E1 -9407.016,E2 -9407.016} C_VEL
LIN {X 0,Y 432.363,Z 401.751,A -85,B 0,C 180,E1 -9408.829,E2 -9408.829} C_VEL
LIN {X 0,Y 433.199,Z 406.77,A -85,B 0,C 180,E1 -9411.94,E2 -9411.94} C_VEL
LIN {X 0,Y 433.616,Z 410.829,A -85,B 0,C 180,E1 -9414.305,E2 -9414.305} C_VEL
LIN {X 0,Y 433.578,Z 413.502,A -85,B 0,C 180,E1 -9415.759,E2 -9415.759} C_VEL
LIN {X 0,Y 433.18,Z 419.165,A -85,B 0,C 180,E1 -9418.724,E2 -9418.724} C_VEL
LIN {X 0,Y 432.802,Z 424.211,A -85,B 0,C 180,E1 -9421.268,E2 -9421.268} C_VEL
LIN {X 0,Y 432.366,Z 431.894,A -85,B 0,C 180,E1 -9425,E2 -9425} C_VEL
LIN {X 0,Y 432.027,Z 439.416,A -85,B 0,C 180,E1 -9428.53,E2 -9428.53} C_VEL
LIN {X 0,Y 431.707,Z 446.964,A -85,B 0,C 180,E1 -9431.982,E2 -9431.982} C_VEL
LIN {X 0,Y 431.656,Z 449.636,A -85,B 0,C 180,E1 -9433.147,E2 -9433.147} C_VEL
LIN {X 0,Y 434.133,Z 462.54,A -85,B 0,C 180,E1 -9433.631,E2 -9433.631} C_VEL
LIN {X 0,Y 435.73,Z 475.234,A -85,B 0,C 180,E1 -9434.266,E2 -9434.266} C_VEL
LIN {X 0,Y 435.081,Z 487.98,A -85,B 0,C 180,E1 -9435.022,E2 -9435.022} C_VEL
LIN {X 0,Y 434.378,Z 498.604,A -85,B 0,C 180,E1 -9435.835,E2 -9435.835} C_VEL
LIN {X 0,Y 433.725,Z 509.475,A -85,B 0,C 180,E1 -9436.888,E2 -9436.888} C_VEL
LIN {X 0,Y 433.073,Z 519.244,A -85,B 0,C 180,E1 -9438.059,E2 -9438.059} C_VEL
LIN {X 0,Y 432.429,Z 527.268,A -85,B 0,C 180,E1 -9439.228,E2 -9439.228} C_VEL
LIN {X 0,Y 431.981,Z 535.159,A -85,B 0,C 180,E1 -9440.637,E2 -9440.637} C_VEL
LIN {X 0,Y 431.627,Z 541.475,A -85,B 0,C 180,E1 -9442.045,E2 -9442.045} C_VEL
LIN {X 0,Y 431.36,Z 547.109,A -85,B 0,C 180,E1 -9443.646,E2 -9443.646} C_VEL
LIN {X 0,Y 431.275,Z 551.501,A -85,B 0,C 180,E1 -9445.326,E2 -9445.326} C_VEL
LIN {X 0,Y 431.189,Z 553.315,A -85,B 0,C 180,E1 -9446.262,E2 -9446.262} C_VEL
LIN {X 0,Y 431.236,Z 554.686,A -85,B 0,C 180,E1 -9447.197,E2 -9447.197} C_VEL
LIN {X 0,Y 431.203,Z 555.661,A -85,B 0,C 180,E1 -9448.132,E2 -9448.132} C_VEL
LIN {X 0,Y 431.169,Z 556.248,A -85,B 0,C 180,E1 -9449.066,E2 -9449.066} C_VEL
LIN {X 0,Y 431.167,Z 556.425,A -85,B 0,C 180,E1 -9450,E2 -9450} C_VEL
LIN {X 0,Y 431.203,Z 555.552,A -85,B 0,C 180,E1 -9451.868,E2 -9451.868} C_VEL
LIN {X 0,Y 431.237,Z 554.534,A -85,B 0,C 180,E1 -9452.802,E2 -9452.802} C_VEL
LIN {X 0,Y 431.19,Z 553.089,A -85,B 0,C 180,E1 -9453.738,E2 -9453.738} C_VEL
LIN {X 0,Y 431.301,Z 550.105,A -85,B 0,C 180,E1 -9455.142,E2 -9455.142} C_VEL
LIN {X 0,Y 431.377,Z 546.062,A -85,B 0,C 180,E1 -9456.548,E2 -9456.548} C_VEL
LIN {X 0,Y 431.657,Z 539.84,A -85,B 0,C 180,E1 -9458.19,E2 -9458.19} C_VEL
LIN {X 0,Y 432.009,Z 533.059,A -85,B 0,C 180,E1 -9459.598,E2 -9459.598} C_VEL
LIN {X 0,Y 432.482,Z 524.631,A -85,B 0,C 180,E1 -9461.007,E2 -9461.007} C_VEL
LIN {X 0,Y 433.089,Z 515.945,A -85,B 0,C 180,E1 -9462.178,E2 -9462.178} C_VEL
LIN {X 0,Y 433.705,Z 505.13,A -85,B 0,C 180,E1 -9463.36,E2 -9463.36} C_VEL
LIN {X 0,Y 434.347,Z 494.579,A -85,B 0,C 180,E1 -9464.285,E2 -9464.285} C_VEL
LIN {X 0,Y 434.967,Z 482.686,A -85,B 0,C 180,E1 -9465.102,E2 -9465.102} C_VEL
LIN {X 0,Y 435.257,Z 474.123,A -85,B 0,C 180,E1 -9465.571,E2 -9465.571} C_VEL
LIN {X 0,Y 433.421,Z 461.036,A -85,B 0,C 180,E1 -9466.176,E2 -9466.176} C_VEL
LIN {X 0,Y 431.646,Z 449.71,A -85,B 0,C 180,E1 -9466.567,E2 -9466.567} C_VEL
LIN {X 0,Y 431.806,Z 442.007,A -85,B 0,C 180,E1 -9469.985,E2 -9469.985} C_VEL
LIN {X 0,Y 432.086,Z 435.359,A -85,B 0,C 180,E1 -9472.977,E2 -9472.977} C_VEL
LIN {X 0,Y 432.344,Z 428.709,A -85,B 0,C 180,E1 -9476.033,E2 -9476.033} C_VEL
LIN {X 0,Y 432.755,Z 420.927,A -85,B 0,C 180,E1 -9479.69,E2 -9479.69} C_VEL
LIN {X 0,Y 433.067,Z 415.238,A -85,B 0,C 180,E1 -9482.448,E2 -9482.448} C_VEL
LIN {X 0,Y 433.337,Z 409.803,A -85,B 0,C 180,E1 -9485.151,E2 -9485.151} C_VEL
LIN {X 0,Y 433.039,Z 405.663,A -85,B 0,C 180,E1 -9487.321,E2 -9487.321} C_VEL
LIN {X 0,Y 432.424,Z 401.622,A -85,B 0,C 180,E1 -9489.635,E2 -9489.635} C_VEL
LIN {X 0,Y 432.361,Z 401.631,A -85,B 0,C 180,E1 -9493.054,E2 -9493.054} C_VEL
LIN {X 0,Y 432.337,Z 401.629,A -85,B 0,C 180,E1 -9495.663,E2 -9495.663} C_VEL
LIN {X 0,Y 432.33,Z 401.631,A -85,B 0,C 180,E1 -9498.397,E2 -9498.397} C_VEL
LIN {X 0,Y 432.342,Z 401.629,A -85,B 0,C 180,E1 -9501.85,E2 -9501.85} C_VEL
LIN {X 0,Y 432.335,Z 401.63,A -85,B 0,C 180,E1 -9505.322,E2 -9505.322} C_VEL
LIN {X 0,Y 432.318,Z 401.636,A -85,B 0,C 180,E1 -9508.653,E2 -9508.653} C_VEL
LIN {X 0,Y 432.374,Z 401.626,A -85,B 0,C 180,E1 -9511.368,E2 -9511.368} C_VEL
LIN {X 0,Y 432.357,Z 401.628,A -85,B 0,C 180,E1 -9513.967,E2 -9513.967} C_VEL
LIN {X 0,Y 432.312,Z 401.634,A -85,B 0,C 180,E1 -9517.035,E2 -9517.035} C_VEL
LIN {X 0,Y 432.379,Z 401.627,A -85,B 0,C 180,E1 -9520.514,E2 -9520.514} C_VEL
LIN {X 0,Y 432.422,Z 401.621,A -85,B 0,C 180,E1 -9523.961,E2 -9523.961} C_VEL
LIN {X 0,Y 432.45,Z 401.617,A -85,B 0,C 180,E1 -9527.803,E2 -9527.803} C_VEL
LIN {X 0,Y 432.483,Z 401.613,A -85,B 0,C 180,E1 -9531.59,E2 -9531.59} C_VEL
LIN {X 0,Y 432.592,Z 401.599,A -85,B 0,C 180,E1 -9534.406,E2 -9534.406} C_VEL
LIN {X 0,Y 432.597,Z 401.599,A -85,B 0,C 180,E1 -9538.138,E2 -9538.138} C_VEL
LIN {X 0,Y 432.726,Z 401.583,A -85,B 0,C 180,E1 -9540,E2 -9540} C_VEL
LIN {X 0,Y 432.599,Z 401.6,A -85,B 0,C 180,E1 -9542.793,E2 -9542.793} C_VEL
LIN {X 0,Y 432.565,Z 401.604,A -85,B 0,C 180,E1 -9546.53,E2 -9546.53} C_VEL
LIN {X 0,Y 432.435,Z 401.618,A -85,B 0,C 180,E1 -9549.353,E2 -9549.353} C_VEL
LIN {X 0,Y 432.436,Z 401.619,A -85,B 0,C 180,E1 -9552.812,E2 -9552.812} C_VEL
LIN {X 0,Y 432.404,Z 401.625,A -85,B 0,C 180,E1 -9556.479,E2 -9556.479} C_VEL
LIN {X 0,Y 432.333,Z 401.632,A -85,B 0,C 180,E1 -9559.961,E2 -9559.961} C_VEL
LIN {X 0,Y 432.313,Z 401.633,A -85,B 0,C 180,E1 -9562.964,E2 -9562.964} C_VEL
LIN {X 0,Y 432.357,Z 401.631,A -85,B 0,C 180,E1 -9566.033,E2 -9566.033} C_VEL
LIN {X 0,Y 432.345,Z 401.629,A -85,B 0,C 180,E1 -9569.187,E2 -9569.187} C_VEL
LIN {X 0,Y 432.324,Z 401.633,A -85,B 0,C 180,E1 -9572.295,E2 -9572.295} C_VEL
LIN {X 0,Y 432.334,Z 401.629,A -85,B 0,C 180,E1 -9574.677,E2 -9574.677} C_VEL
LIN {X 0,Y 432.347,Z 401.63,A -85,B 0,C 180,E1 -9578.149,E2 -9578.149} C_VEL
LIN {X 0,Y 432.367,Z 401.63,A -85,B 0,C 180,E1 -9581.609,E2 -9581.609} C_VEL
LIN {X 0,Y 432.373,Z 401.624,A -85,B 0,C 180,E1 -9584.342,E2 -9584.342} C_VEL
LIN {X 0,Y 432.361,Z 401.626,A -85,B 0,C 180,E1 -9587.01,E2 -9587.01} C_VEL
LIN {X 0,Y 432.353,Z 401.629,A -85,B 0,C 180,E1 -9589.818,E2 -9589.818} C_VEL
LIN {X 0,Y 432.313,Z 401.633,A -85,B 0,C 180,E1 -9593.024,E2 -9593.024} C_VEL
LIN {X 0,Y 432.356,Z 401.626,A -85,B 0,C 180,E1 -9595.997,E2 -9595.997} C_VEL
LIN {X 0,Y 432.345,Z 401.631,A -85,B 0,C 180,E1 -9599.49,E2 -9599.49} C_VEL
LIN {X 0,Y 432.391,Z 401.625,A -85,B 0,C 180,E1 -9602.929,E2 -9602.929} C_VEL
LIN {X 0,Y 432.369,Z 401.625,A -85,B 0,C 180,E1 -9606.024,E2 -9606.024} C_VEL
LIN {X 0,Y 432.168,Z 401.656,A -85,B 0,C 180,E1 -9609.037,E2 -9609.037} C_VEL
LIN {X 0,Y 432.163,Z 404.056,A -85,B 0,C 180,E1 -9611.02,E2 -9611.02} C_VEL
LIN {X 0,Y 432.057,Z 408.022,A -85,B 0,C 180,E1 -9613.947,E2 -9613.947} C_VEL
LIN {X 0,Y 431.949,Z 413.344,A -85,B 0,C 180,E1 -9617.789,E2 -9617.789} C_VEL
LIN {X 0,Y 431.78,Z 418.728,A -85,B 0,C 180,E1 -9621.577,E2 -9621.577} C_VEL
LIN {X 0,Y 431.789,Z 421.432,A -85,B 0,C 180,E1 -9623.458,E2 -9623.458} C_VEL
LIN {X 0,Y 431.678,Z 425.521,A -85,B 0,C 180,E1 -9626.266,E2 -9626.266} C_VEL
LIN {X 0,Y 431.545,Z 427.386,A -85,B 0,C 180,E1 -9627.521,E2 -9627.521} C_VEL
LIN {X 0,Y 434.314,Z 441.376,A -85,B 0,C 180,E1 -9628.073,E2 -9628.073} C_VEL
LIN {X 0,Y 435.648,Z 448.732,A -85,B 0,C 180,E1 -9628.44,E2 -9628.44} C_VEL
LIN {X 0,Y 435.203,Z 460.239,A -85,B 0,C 180,E1 -9629.075,E2 -9629.075} C_VEL
LIN {X 0,Y 434.548,Z 471.54,A -85,B 0,C 180,E1 -9629.884,E2 -9629.884} C_VEL
LIN {X 0,Y 434.164,Z 478.66,A -85,B 0,C 180,E1 -9630.503,E2 -9630.503} C_VEL
LIN {X 0,Y 433.262,Z 483.43,A -85,B 0,C 180,E1 -9630.949,E2 -9630.949} C_VEL
LIN {X 0,Y 429.955,Z 490.881,A -85,B 0,C 180,E1 -9631.702,E2 -9631.702} C_VEL
LIN {X 0,Y 426.602,Z 497.794,A -85,B 0,C 180,E1 -9632.543,E2 -9632.543} C_VEL
LIN {X 0,Y 425.64,Z 501.721,A -85,B 0,C 180,E1 -9633.124,E2 -9633.124} C_VEL
LIN {X 0,Y 425.113,Z 509.579,A -85,B 0,C 180,E1 -9634.504,E2 -9634.504} C_VEL
LIN {X 0,Y 424.807,Z 515.136,A -85,B 0,C 180,E1 -9635.697,E2 -9635.697} C_VEL
LIN {X 0,Y 424.592,Z 520.404,A -85,B 0,C 180,E1 -9637.083,E2 -9637.083} C_VEL
LIN {X 0,Y 424.322,Z 524.836,A -85,B 0,C 180,E1 -9638.573,E2 -9638.573} C_VEL
LIN {X 0,Y 424.209,Z 527.103,A -85,B 0,C 180,E1 -9639.536,E2 -9639.536} C_VEL
LIN {X 0,Y 424.14,Z 528.888,A -85,B 0,C 180,E1 -9640.502,E2 -9640.502} C_VEL
LIN {X 0,Y 424.09,Z 530.91,A -85,B 0,C 180,E1 -9642.111,E2 -9642.111} C_VEL
LIN {X 0,Y 423.976,Z 531.736,A -85,B 0,C 180,E1 -9643.419,E2 -9643.419} C_VEL
LIN {X 0,Y 423.96,Z 531.828,A -85,B 0,C 180,E1 -9644.398,E2 -9644.398} C_VEL
LIN {X 0,Y 424.02,Z 531.117,A -85,B 0,C 180,E1 -9645.986,E2 -9645.986} C_VEL
LIN {X 0,Y 424.066,Z 529.627,A -85,B 0,C 180,E1 -9647.356,E2 -9647.356} C_VEL
LIN {X 0,Y 424.325,Z 526.125,A -85,B 0,C 180,E1 -9649.252,E2 -9649.252} C_VEL
LIN {X 0,Y 424.581,Z 521.829,A -85,B 0,C 180,E1 -9650.847,E2 -9650.847} C_VEL
LIN {X 0,Y 424.916,Z 516.439,A -85,B 0,C 180,E1 -9652.359,E2 -9652.359} C_VEL
LIN {X 0,Y 425.429,Z 509.545,A -85,B 0,C 180,E1 -9653.874,E2 -9653.874} C_VEL
LIN {X 0,Y 425.968,Z 502.077,A -85,B 0,C 180,E1 -9655.2,E2 -9655.2} C_VEL
LIN {X 0,Y 426.566,Z 493.745,A -85,B 0,C 180,E1 -9656.413,E2 -9656.413} C_VEL
LIN {X 0,Y 427.329,Z 484.167,A -85,B 0,C 180,E1 -9657.552,E2 -9657.552} C_VEL
LIN {X 0,Y 428.088,Z 473.563,A -85,B 0,C 180,E1 -9658.564,E2 -9658.564} C_VEL
LIN {X 0,Y 428.788,Z 461.842,A -85,B 0,C 180,E1 -9659.453,E2 -9659.453} C_VEL
LIN {X 0,Y 429.359,Z 449.854,A -85,B 0,C 180,E1 -9660.15,E2 -9660.15} C_VEL
LIN {X 0,Y 426.879,Z 437.458,A -85,B 0,C 180,E1 -9660.805,E2 -9660.805} C_VEL
LIN {X 0,Y 424.424,Z 427.762,A -85,B 0,C 180,E1 -9661.24,E2 -9661.24} C_VEL
LIN {X 0,Y 424.529,Z 423.56,A -85,B 0,C 180,E1 -9664.253,E2 -9664.253} C_VEL
LIN {X 0,Y 424.727,Z 418.797,A -85,B 0,C 180,E1 -9667.751,E2 -9667.751} C_VEL
LIN {X 0,Y 424.861,Z 415.211,A -85,B 0,C 180,E1 -9670.454,E2 -9670.454} C_VEL
LIN {X 0,Y 425.035,Z 411.493,A -85,B 0,C 180,E1 -9673.319,E2 -9673.319} C_VEL
LIN {X 0,Y 425.211,Z 407.319,A -85,B 0,C 180,E1 -9676.655,E2 -9676.655} C_VEL
LIN {X 0,Y 425.328,Z 403.892,A -85,B 0,C 180,E1 -9679.471,E2 -9679.471} C_VEL
LIN {X 0,Y 425.265,Z 402.515,A -85,B 0,C 180,E1 -9681.098,E2 -9681.098} C_VEL
LIN {X 0,Y 425.296,Z 402.514,A -85,B 0,C 180,E1 -9684.664,E2 -9684.664} C_VEL
LIN {X 0,Y 425.267,Z 402.516,A -85,B 0,C 180,E1 -9688.073,E2 -9688.073} C_VEL
LIN {X 0,Y 425.333,Z 402.506,A -85,B 0,C 180,E1 -9691.368,E2 -9691.368} C_VEL
LIN {X 0,Y 425.29,Z 402.51,A -85,B 0,C 180,E1 -9694.554,E2 -9694.554} C_VEL
LIN {X 0,Y 425.282,Z 402.509,A -85,B 0,C 180,E1 -9697.661,E2 -9697.661} C_VEL
LIN {X 0,Y 425.356,Z 402.5,A -85,B 0,C 180,E1 -9700.704,E2 -9700.704} C_VEL
LIN {X 0,Y 425.382,Z 402.497,A -85,B 0,C 180,E1 -9703.688,E2 -9703.688} C_VEL
LIN {X 0,Y 425.406,Z 402.498,A -85,B 0,C 180,E1 -9707.598,E2 -9707.598} C_VEL
LIN {X 0,Y 425.436,Z 402.49,A -85,B 0,C 180,E1 -9711.45,E2 -9711.45} C_VEL
LIN {X 0,Y 425.548,Z 402.477,A -85,B 0,C 180,E1 -9714.313,E2 -9714.313} C_VEL
LIN {X 0,Y 425.57,Z 402.477,A -85,B 0,C 180,E1 -9718.107,E2 -9718.107} C_VEL
LIN {X 0,Y 425.696,Z 402.459,A -85,B 0,C 180,E1 -9720,E2 -9720} C_VEL
LIN {X 0,Y 425.552,Z 402.477,A -85,B 0,C 180,E1 -9722.84,E2 -9722.84} C_VEL
LIN {X 0,Y 425.525,Z 402.48,A -85,B 0,C 180,E1 -9726.639,E2 -9726.639} C_VEL
LIN {X 0,Y 425.398,Z 402.496,A -85,B 0,C 180,E1 -9729.51,E2 -9729.51} C_VEL
LIN {X 0,Y 425.399,Z 402.498,A -85,B 0,C 180,E1 -9732.911,E2 -9732.911} C_VEL
LIN {X 0,Y 425.365,Z 402.501,A -85,B 0,C 180,E1 -9736.609,E2 -9736.609} C_VEL
LIN {X 0,Y 425.323,Z 402.506,A -85,B 0,C 180,E1 -9739.636,E2 -9739.636} C_VEL
LIN {X 0,Y 425.302,Z 402.512,A -85,B 0,C 180,E1 -9743.366,E2 -9743.366} C_VEL
LIN {X 0,Y 425.344,Z 402.504,A -85,B 0,C 180,E1 -9746.845,E2 -9746.845} C_VEL
LIN {X 0,Y 425.314,Z 402.508,A -85,B 0,C 180,E1 -9749.718,E2 -9749.718} C_VEL
LIN {X 0,Y 425.279,Z 402.511,A -85,B 0,C 180,E1 -9753.049,E2 -9753.049} C_VEL
LIN {X 0,Y 425.281,Z 402.508,A -85,B 0,C 180,E1 -9755.93,E2 -9755.93} C_VEL
LIN {X 0,Y 425.293,Z 402.506,A -85,B 0,C 180,E1 -9759.044,E2 -9759.044} C_VEL
LIN {X 0,Y 425.272,Z 402.514,A -85,B 0,C 180,E1 -9762.654,E2 -9762.654} C_VEL
LIN {X 0,Y 425.267,Z 402.514,A -85,B 0,C 180,E1 -9766.046,E2 -9766.046} C_VEL
LIN {X 0,Y 425.311,Z 402.613,A -85,B 0,C 180,E1 -9768.482,E2 -9768.482} C_VEL
LIN {X 0,Y 426.059,Z 406.834,A -85,B 0,C 180,E1 -9771.185,E2 -9771.185} C_VEL
LIN {X 0,Y 426.61,Z 411.245,A -85,B 0,C 180,E1 -9773.826,E2 -9773.826} C_VEL
LIN {X 0,Y 426.523,Z 415.015,A -85,B 0,C 180,E1 -9775.929,E2 -9775.929} C_VEL
LIN {X 0,Y 426.068,Z 421.252,A -85,B 0,C 180,E1 -9779.247,E2 -9779.247} C_VEL
LIN {X 0,Y 425.587,Z 427.589,A -85,B 0,C 180,E1 -9782.459,E2 -9782.459} C_VEL
LIN {X 0,Y 425.231,Z 433.971,A -85,B 0,C 180,E1 -9785.595,E2 -9785.595} C_VEL
LIN {X 0,Y 424.947,Z 440.401,A -85,B 0,C 180,E1 -9788.664,E2 -9788.664} C_VEL
LIN {X 0,Y 424.637,Z 447.94,A -85,B 0,C 180,E1 -9792.171,E2 -9792.171} C_VEL
LIN {X 0,Y 424.618,Z 449.426,A -85,B 0,C 180,E1 -9792.818,E2 -9792.818} C_VEL
LIN {X 0,Y 427.161,Z 462.285,A -85,B 0,C 180,E1 -9793.317,E2 -9793.317} C_VEL
LIN {X 0,Y 428.839,Z 475.627,A -85,B 0,C 180,E1 -9794.007,E2 -9794.007} C_VEL
LIN {X 0,Y 428.256,Z 488.228,A -85,B 0,C 180,E1 -9794.777,E2 -9794.777} C_VEL
LIN {X 0,Y 427.405,Z 500.042,A -85,B 0,C 180,E1 -9795.721,E2 -9795.721} C_VEL
LIN {X 0,Y 426.73,Z 510.612,A -85,B 0,C 180,E1 -9796.791,E2 -9796.791} C_VEL
LIN {X 0,Y 425.979,Z 521.008,A -85,B 0,C 180,E1 -9798.099,E2 -9798.099} C_VEL
LIN {X 0,Y 425.263,Z 530.043,A -85,B 0,C 180,E1 -9799.526,E2 -9799.526} C_VEL
LIN {X 0,Y 424.815,Z 537.34,A -85,B 0,C 180,E1 -9800.958,E2 -9800.958} C_VEL
LIN {X 0,Y 424.478,Z 543.2,A -85,B 0,C 180,E1 -9802.389,E2 -9802.389} C_VEL
LIN {X 0,Y 424.249,Z 547.451,A -85,B 0,C 180,E1 -9803.693,E2 -9803.693} C_VEL
LIN {X 0,Y 424.204,Z 551.355,A -85,B 0,C 180,E1 -9805.248,E2 -9805.248} C_VEL
LIN {X 0,Y 424.101,Z 553.15,A -85,B 0,C 180,E1 -9806.199,E2 -9806.199} C_VEL
LIN {X 0,Y 424.132,Z 554.51,A -85,B 0,C 180,E1 -9807.15,E2 -9807.15} C_VEL
LIN {X 0,Y 424.129,Z 555.478,A -85,B 0,C 180,E1 -9808.101,E2 -9808.101} C_VEL
LIN {X 0,Y 424.088,Z 556.056,A -85,B 0,C 180,E1 -9809.05,E2 -9809.05} C_VEL
LIN {X 0,Y 424.084,Z 556.217,A -85,B 0,C 180,E1 -9810,E2 -9810} C_VEL
LIN {X 0,Y 424.129,Z 555.328,A -85,B 0,C 180,E1 -9811.899,E2 -9811.899} C_VEL
LIN {X 0,Y 424.134,Z 554.3,A -85,B 0,C 180,E1 -9812.849,E2 -9812.849} C_VEL
LIN {X 0,Y 424.101,Z 552.838,A -85,B 0,C 180,E1 -9813.8,E2 -9813.8} C_VEL
LIN {X 0,Y 424.214,Z 549.836,A -85,B 0,C 180,E1 -9815.228,E2 -9815.228} C_VEL
LIN {X 0,Y 424.301,Z 545.771,A -85,B 0,C 180,E1 -9816.658,E2 -9816.658} C_VEL
LIN {X 0,Y 424.605,Z 539.518,A -85,B 0,C 180,E1 -9818.327,E2 -9818.327} C_VEL
LIN {X 0,Y 424.96,Z 532.703,A -85,B 0,C 180,E1 -9819.759,E2 -9819.759} C_VEL
LIN {X 0,Y 425.49,Z 524.222,A -85,B 0,C 180,E1 -9821.191,E2 -9821.191} C_VEL
LIN {X 0,Y 426.104,Z 515.481,A -85,B 0,C 180,E1 -9822.381,E2 -9822.381} C_VEL
LIN {X 0,Y 426.736,Z 504.464,A -85,B 0,C 180,E1 -9823.598,E2 -9823.598} C_VEL
LIN {X 0,Y 427.423,Z 493.986,A -85,B 0,C 180,E1 -9824.521,E2 -9824.521} C_VEL
LIN {X 0,Y 428.065,Z 481.951,A -85,B 0,C 180,E1 -9825.351,E2 -9825.351} C_VEL
LIN {X 0,Y 428.274,Z 474.445,A -85,B 0,C 180,E1 -9825.77,E2 -9825.77} C_VEL
LIN {X 0,Y 426.453,Z 461.355,A -85,B 0,C 180,E1 -9826.398,E2 -9826.398} C_VEL
LIN {X 0,Y 424.565,Z 449.508,A -85,B 0,C 180,E1 -9826.82,E2 -9826.82} C_VEL
LIN {X 0,Y 424.783,Z 441.741,A -85,B 0,C 180,E1 -9830.33,E2 -9830.33} C_VEL
LIN {X 0,Y 425.054,Z 435.114,A -85,B 0,C 180,E1 -9833.379,E2 -9833.379} C_VEL
LIN {X 0,Y 425.31,Z 428.452,A -85,B 0,C 180,E1 -9836.497,E2 -9836.497} C_VEL
LIN {X 0,Y 425.713,Z 421.802,A -85,B 0,C 180,E1 -9839.686,E2 -9839.686} C_VEL
LIN {X 0,Y 426.043,Z 415.639,A -85,B 0,C 180,E1 -9842.722,E2 -9842.722} C_VEL
LIN {X 0,Y 426.331,Z 410.696,A -85,B 0,C 180,E1 -9845.237,E2 -9845.237} C_VEL
LIN {X 0,Y 426.101,Z 407.33,A -85,B 0,C 180,E1 -9847.014,E2 -9847.014} C_VEL
LIN {X 0,Y 425.367,Z 402.501,A -85,B 0,C 180,E1 -9849.701,E2 -9849.701} C_VEL
LIN {X 0,Y 425.312,Z 402.506,A -85,B 0,C 180,E1 -9853.358,E2 -9853.358} C_VEL
LIN {X 0,Y 425.26,Z 402.513,A -85,B 0,C 180,E1 -9856.647,E2 -9856.647} C_VEL
LIN {X 0,Y 425.285,Z 402.508,A -85,B 0,C 180,E1 -9859.872,E2 -9859.872} C_VEL
LIN {X 0,Y 425.279,Z 402.51,A -85,B 0,C 180,E1 -9862.486,E2 -9862.486} C_VEL
LIN {X 0,Y 425.302,Z 402.506,A -85,B 0,C 180,E1 -9865.817,E2 -9865.817} C_VEL
LIN {X 0,Y 425.294,Z 402.508,A -85,B 0,C 180,E1 -9869.236,E2 -9869.236} C_VEL
LIN {X 0,Y 425.343,Z 402.504,A -85,B 0,C 180,E1 -9872.442,E2 -9872.442} C_VEL
LIN {X 0,Y 425.344,Z 402.501,A -85,B 0,C 180,E1 -9875.601,E2 -9875.601} C_VEL
LIN {X 0,Y 425.286,Z 402.51,A -85,B 0,C 180,E1 -9878.681,E2 -9878.681} C_VEL
LIN {X 0,Y 425.325,Z 402.504,A -85,B 0,C 180,E1 -9881.702,E2 -9881.702} C_VEL
LIN {X 0,Y 425.34,Z 402.503,A -85,B 0,C 180,E1 -9884.67,E2 -9884.67} C_VEL
LIN {X 0,Y 425.403,Z 402.494,A -85,B 0,C 180,E1 -9887.598,E2 -9887.598} C_VEL
LIN {X 0,Y 425.434,Z 402.49,A -85,B 0,C 180,E1 -9891.45,E2 -9891.45} C_VEL
LIN {X 0,Y 425.567,Z 402.475,A -85,B 0,C 180,E1 -9894.313,E2 -9894.313} C_VEL
LIN {X 0,Y 425.567,Z 402.475,A -85,B 0,C 180,E1 -9898.107,E2 -9898.107} C_VEL
LIN {X 0,Y 425.696,Z 402.459,A -85,B 0,C 180,E1 -9900,E2 -9900} C_VEL
LIN {X 0,Y 425.551,Z 402.477,A -85,B 0,C 180,E1 -9902.84,E2 -9902.84} C_VEL
LIN {X 0,Y 425.523,Z 402.482,A -85,B 0,C 180,E1 -9906.642,E2 -9906.642} C_VEL
LIN {X 0,Y 425.394,Z 402.496,A -85,B 0,C 180,E1 -9909.509,E2 -9909.509} C_VEL
LIN {X 0,Y 425.395,Z 402.495,A -85,B 0,C 180,E1 -9912.91,E2 -9912.91} C_VEL
LIN {X 0,Y 425.353,Z 402.502,A -85,B 0,C 180,E1 -9916.605,E2 -9916.605} C_VEL
LIN {X 0,Y 425.32,Z 402.505,A -85,B 0,C 180,E1 -9919.636,E2 -9919.636} C_VEL
LIN {X 0,Y 425.3,Z 402.507,A -85,B 0,C 180,E1 -9923.365,E2 -9923.365} C_VEL
LIN {X 0,Y 425.341,Z 402.501,A -85,B 0,C 180,E1 -9926.845,E2 -9926.845} C_VEL
LIN {X 0,Y 425.311,Z 402.507,A -85,B 0,C 180,E1 -9929.718,E2 -9929.718} C_VEL
LIN {X 0,Y 425.277,Z 402.509,A -85,B 0,C 180,E1 -9933.048,E2 -9933.048} C_VEL
LIN {X 0,Y 425.278,Z 402.513,A -85,B 0,C 180,E1 -9935.93,E2 -9935.93} C_VEL
LIN {X 0,Y 425.307,Z 402.505,A -85,B 0,C 180,E1 -9939.047,E2 -9939.047} C_VEL
LIN {X 0,Y 425.326,Z 402.502,A -85,B 0,C 180,E1 -9942.647,E2 -9942.647} C_VEL
LIN {X 0,Y 425.314,Z 402.505,A -85,B 0,C 180,E1 -9946.052,E2 -9946.052} C_VEL
LIN {X 0,Y 425.305,Z 402.504,A -85,B 0,C 180,E1 -9948.626,E2 -9948.626} C_VEL
LIN {X 0,Y 425.319,Z 402.504,A -85,B 0,C 180,E1 -9951.105,E2 -9951.105} C_VEL
LIN {X 0,Y 425.297,Z 402.505,A -85,B 0,C 180,E1 -9954.665,E2 -9954.665} C_VEL
LIN {X 0,Y 425.262,Z 402.509,A -85,B 0,C 180,E1 -9958.074,E2 -9958.074} C_VEL
LIN {X 0,Y 425.329,Z 402.506,A -85,B 0,C 180,E1 -9961.369,E2 -9961.369} C_VEL
LIN {X 0,Y 425.294,Z 402.506,A -85,B 0,C 180,E1 -9964.555,E2 -9964.555} C_VEL
LIN {X 0,Y 425.277,Z 402.509,A -85,B 0,C 180,E1 -9966.634,E2 -9966.634} C_VEL
LIN {X 0,Y 425.149,Z 402.526,A -85,B 0,C 180,E1 -9968.675,E2 -9968.675} C_VEL
LIN {X 0,Y 425.117,Z 403.135,A -85,B 0,C 180,E1 -9969.686,E2 -9969.686} C_VEL
LIN {X 0,Y 424.999,Z 407.111,A -85,B 0,C 180,E1 -9972.684,E2 -9972.684} C_VEL
LIN {X 0,Y 424.884,Z 411.101,A -85,B 0,C 180,E1 -9975.634,E2 -9975.634} C_VEL
LIN {X 0,Y 424.919,Z 413.789,A -85,B 0,C 180,E1 -9977.584,E2 -9977.584} C_VEL
LIN {X 0,Y 424.716,Z 419.184,A -85,B 0,C 180,E1 -9981.436,E2 -9981.436} C_VEL
LIN {X 0,Y 424.72,Z 421.888,A -85,B 0,C 180,E1 -9983.349,E2 -9983.349} C_VEL
LIN {X 0,Y 424.616,Z 426.015,A -85,B 0,C 180,E1 -9986.204,E2 -9986.204} C_VEL
LIN {X 0,Y 424.544,Z 427.565,A -85,B 0,C 180,E1 -9987.272,E2 -9987.272} C_VEL
LIN {X 0,Y 427.258,Z 441.574,A -85,B 0,C 180,E1 -9987.835,E2 -9987.835} C_VEL
LIN {X 0,Y 428.731,Z 450.553,A -85,B 0,C 180,E1 -9988.298,E2 -9988.298} C_VEL
LIN {X 0,Y 428.132,Z 463.427,A -85,B 0,C 180,E1 -9989.06,E2 -9989.06} C_VEL
LIN {X 0,Y 427.498,Z 474.142,A -85,B 0,C 180,E1 -9989.882,E2 -9989.882} C_VEL
LIN {X 0,Y 426.808,Z 485.079,A -85,B 0,C 180,E1 -9990.944,E2 -9990.944} C_VEL
LIN {X 0,Y 426.152,Z 494.864,A -85,B 0,C 180,E1 -9992.127,E2 -9992.127} C_VEL
LIN {X 0,Y 425.64,Z 501.721,A -85,B 0,C 180,E1 -9993.124,E2 -9993.124} C_VEL
LIN {X 0,Y 424.726,Z 505.492,A -85,B 0,C 180,E1 -9993.73,E2 -9993.73} C_VEL
LIN {X 0,Y 421.558,Z 511.192,A -85,B 0,C 180,E1 -9994.742,E2 -9994.742} C_VEL
LIN {X 0,Y 418.441,Z 516.246,A -85,B 0,C 180,E1 -9995.822,E2 -9995.822} C_VEL
LIN {X 0,Y 417.614,Z 518.974,A -85,B 0,C 180,E1 -9996.528,E2 -9996.528} C_VEL
LIN {X 0,Y 417.274,Z 524.32,A -85,B 0,C 180,E1 -9998.231,E2 -9998.231} C_VEL
LIN {X 0,Y 417.094,Z 527.719,A -85,B 0,C 180,E1 -9999.701,E2 -9999.701} C_VEL
LIN {X 0,Y 417.048,Z 529.405,A -85,B 0,C 180,E1 -10000.683,E2 -10000.683} C_VEL
LIN {X 0,Y 417.001,Z 531.167,A -85,B 0,C 180,E1 -10002.174,E2 -10002.174} C_VEL
LIN {X 0,Y 416.879,Z 531.979,A -85,B 0,C 180,E1 -10003.652,E2 -10003.652} C_VEL
LIN {X 0,Y 416.88,Z 531.999,A -85,B 0,C 180,E1 -10004.648,E2 -10004.648} C_VEL
LIN {X 0,Y 416.939,Z 531.285,A -85,B 0,C 180,E1 -10006.095,E2 -10006.095} C_VEL
LIN {X 0,Y 417.013,Z 529.513,A -85,B 0,C 180,E1 -10007.659,E2 -10007.659} C_VEL
LIN {X 0,Y 417.277,Z 526.254,A -85,B 0,C 180,E1 -10009.407,E2 -10009.407} C_VEL
LIN {X 0,Y 417.59,Z 521.333,A -85,B 0,C 180,E1 -10011.213,E2 -10011.213} C_VEL
LIN {X 0,Y 417.995,Z 515.748,A -85,B 0,C 180,E1 -10012.75,E2 -10012.75} C_VEL
LIN {X 0,Y 418.514,Z 508.653,A -85,B 0,C 180,E1 -10014.294,E2 -10014.294} C_VEL
LIN {X 0,Y 419.136,Z 501.159,A -85,B 0,C 180,E1 -10015.608,E2 -10015.608} C_VEL
LIN {X 0,Y 419.791,Z 492.325,A -85,B 0,C 180,E1 -10016.873,E2 -10016.873} C_VEL
LIN {X 0,Y 420.66,Z 482.333,A -85,B 0,C 180,E1 -10018.026,E2 -10018.026} C_VEL
LIN {X 0,Y 421.403,Z 471.255,A -85,B 0,C 180,E1 -10019.06,E2 -10019.06} C_VEL
LIN {X 0,Y 422.175,Z 459.848,A -85,B 0,C 180,E1 -10019.892,E2 -10019.892} C_VEL
LIN {X 0,Y 422.494,Z 450.386,A -85,B 0,C 180,E1 -10020.442,E2 -10020.442} C_VEL
LIN {X 0,Y 419.931,Z 437.751,A -85,B 0,C 180,E1 -10021.129,E2 -10021.129} C_VEL
LIN {X 0,Y 417.368,Z 427.994,A -85,B 0,C 180,E1 -10021.572,E2 -10021.572} C_VEL
LIN {X 0,Y 417.471,Z 423.419,A -85,B 0,C 180,E1 -10024.916,E2 -10024.916} C_VEL
LIN {X 0,Y 417.695,Z 419.626,A -85,B 0,C 180,E1 -10027.739,E2 -10027.739} C_VEL
LIN {X 0,Y 417.844,Z 415.393,A -85,B 0,C 180,E1 -10030.992,E2 -10030.992} C_VEL
LIN {X 0,Y 417.993,Z 411.953,A -85,B 0,C 180,E1 -10033.698,E2 -10033.698} C_VEL
LIN {X 0,Y 418.151,Z 408.56,A -85,B 0,C 180,E1 -10036.441,E2 -10036.441} C_VEL
LIN {X 0,Y 418.303,Z 405.357,A -85,B 0,C 180,E1 -10039.117,E2 -10039.117} C_VEL
LIN {X 0,Y 418.209,Z 403.61,A -85,B 0,C 180,E1 -10040.626,E2 -10040.626} C_VEL
LIN {X 0,Y 418.237,Z 403.393,A -85,B 0,C 180,E1 -10042.776,E2 -10042.776} C_VEL
LIN {X 0,Y 418.245,Z 403.391,A -85,B 0,C 180,E1 -10046.323,E2 -10046.323} C_VEL
LIN {X 0,Y 418.257,Z 403.388,A -85,B 0,C 180,E1 -10049.729,E2 -10049.729} C_VEL
LIN {X 0,Y 418.299,Z 403.381,A -85,B 0,C 180,E1 -10053.023,E2 -10053.023} C_VEL
LIN {X 0,Y 418.271,Z 403.383,A -85,B 0,C 180,E1 -10056.218,E2 -10056.218} C_VEL
LIN {X 0,Y 418.244,Z 403.387,A -85,B 0,C 180,E1 -10059.337,E2 -10059.337} C_VEL
LIN {X 0,Y 418.282,Z 403.381,A -85,B 0,C 180,E1 -10062.396,E2 -10062.396} C_VEL
LIN {X 0,Y 418.297,Z 403.379,A -85,B 0,C 180,E1 -10065.403,E2 -10065.403} C_VEL
LIN {X 0,Y 418.311,Z 403.377,A -85,B 0,C 180,E1 -10068.369,E2 -10068.369} C_VEL
LIN {X 0,Y 418.507,Z 403.356,A -85,B 0,C 180,E1 -10072.279,E2 -10072.279} C_VEL
LIN {X 0,Y 418.507,Z 403.354,A -85,B 0,C 180,E1 -10074.217,E2 -10074.217} C_VEL
LIN {X 0,Y 418.539,Z 403.353,A -85,B 0,C 180,E1 -10078.076,E2 -10078.076} C_VEL
LIN {X 0,Y 418.666,Z 403.335,A -85,B 0,C 180,E1 -10080,E2 -10080} C_VEL
LIN {X 0,Y 418.506,Z 403.355,A -85,B 0,C 180,E1 -10082.888,E2 -10082.888} C_VEL
LIN {X 0,Y 418.488,Z 403.357,A -85,B 0,C 180,E1 -10086.751,E2 -10086.751} C_VEL
LIN {X 0,Y 418.354,Z 403.374,A -85,B 0,C 180,E1 -10089.671,E2 -10089.671} C_VEL
LIN {X 0,Y 418.35,Z 403.377,A -85,B 0,C 180,E1 -10093.007,E2 -10093.007} C_VEL
LIN {X 0,Y 418.315,Z 403.379,A -85,B 0,C 180,E1 -10096.739,E2 -10096.739} C_VEL
LIN {X 0,Y 418.266,Z 403.386,A -85,B 0,C 180,E1 -10099.791,E2 -10099.791} C_VEL
LIN {X 0,Y 418.233,Z 403.39,A -85,B 0,C 180,E1 -10102.737,E2 -10102.737} C_VEL
LIN {X 0,Y 418.267,Z 403.385,A -85,B 0,C 180,E1 -10105.905,E2 -10105.905} C_VEL
LIN {X 0,Y 418.271,Z 403.386,A -85,B 0,C 180,E1 -10109.162,E2 -10109.162} C_VEL
LIN {X 0,Y 418.254,Z 403.387,A -85,B 0,C 180,E1 -10112.845,E2 -10112.845} C_VEL
LIN {X 0,Y 418.245,Z 403.384,A -85,B 0,C 180,E1 -10116.239,E2 -10116.239} C_VEL
LIN {X 0,Y 418.247,Z 403.386,A -85,B 0,C 180,E1 -10119.683,E2 -10119.683} C_VEL
LIN {X 0,Y 418.227,Z 403.39,A -85,B 0,C 180,E1 -10122.322,E2 -10122.322} C_VEL
LIN {X 0,Y 418.237,Z 403.389,A -85,B 0,C 180,E1 -10125.11,E2 -10125.11} C_VEL
LIN {X 0,Y 418.271,Z 403.439,A -85,B 0,C 180,E1 -10128.096,E2 -10128.096} C_VEL
LIN {X 0,Y 418.894,Z 407.114,A -85,B 0,C 180,E1 -10130.513,E2 -10130.513} C_VEL
LIN {X 0,Y 419.574,Z 411.963,A -85,B 0,C 180,E1 -10133.516,E2 -10133.516} C_VEL
LIN {X 0,Y 419.526,Z 416.064,A -85,B 0,C 180,E1 -10135.862,E2 -10135.862} C_VEL
LIN {X 0,Y 419.121,Z 421.447,A -85,B 0,C 180,E1 -10138.781,E2 -10138.781} C_VEL
LIN {X 0,Y 418.593,Z 427.561,A -85,B 0,C 180,E1 -10141.959,E2 -10141.959} C_VEL
LIN {X 0,Y 418.229,Z 433.911,A -85,B 0,C 180,E1 -10145.159,E2 -10145.159} C_VEL
LIN {X 0,Y 417.879,Z 441.399,A -85,B 0,C 180,E1 -10148.802,E2 -10148.802} C_VEL
LIN {X 0,Y 417.556,Z 449.119,A -85,B 0,C 180,E1 -10152.463,E2 -10152.463} C_VEL
LIN {X 0,Y 420.32,Z 462.892,A -85,B 0,C 180,E1 -10153.03,E2 -10153.03} C_VEL
LIN {X 0,Y 421.968,Z 476.144,A -85,B 0,C 180,E1 -10153.739,E2 -10153.739} C_VEL
LIN {X 0,Y 421.429,Z 488.559,A -85,B 0,C 180,E1 -10154.525,E2 -10154.525} C_VEL
LIN {X 0,Y 420.531,Z 500.225,A -85,B 0,C 180,E1 -10155.482,E2 -10155.482} C_VEL
LIN {X 0,Y 419.806,Z 510.715,A -85,B 0,C 180,E1 -10156.569,E2 -10156.569} C_VEL
LIN {X 0,Y 419.168,Z 519.308,A -85,B 0,C 180,E1 -10157.656,E2 -10157.656} C_VEL
LIN {X 0,Y 418.455,Z 527.244,A -85,B 0,C 180,E1 -10158.864,E2 -10158.864} C_VEL
LIN {X 0,Y 417.917,Z 535.039,A -85,B 0,C 180,E1 -10160.319,E2 -10160.319} C_VEL
LIN {X 0,Y 417.519,Z 541.293,A -85,B 0,C 180,E1 -10161.774,E2 -10161.774} C_VEL
LIN {X 0,Y 417.236,Z 546.28,A -85,B 0,C 180,E1 -10163.228,E2 -10163.228} C_VEL
LIN {X 0,Y 417.129,Z 550.146,A -85,B 0,C 180,E1 -10164.683,E2 -10164.683} C_VEL
LIN {X 0,Y 417.016,Z 552.991,A -85,B 0,C 180,E1 -10166.135,E2 -10166.135} C_VEL
LIN {X 0,Y 417.056,Z 555.299,A -85,B 0,C 180,E1 -10168.068,E2 -10168.068} C_VEL
LIN {X 0,Y 417.011,Z 555.867,A -85,B 0,C 180,E1 -10169.034,E2 -10169.034} C_VEL
LIN {X 0,Y 417.004,Z 556.007,A -85,B 0,C 180,E1 -10170,E2 -10170} C_VEL
LIN {X 0,Y 417.057,Z 555.098,A -85,B 0,C 180,E1 -10171.931,E2 -10171.931} C_VEL
LIN {X 0,Y 417.031,Z 554.059,A -85,B 0,C 180,E1 -10172.898,E2 -10172.898} C_VEL
LIN {X 0,Y 417.017,Z 552.575,A -85,B 0,C 180,E1 -10173.865,E2 -10173.865} C_VEL
LIN {X 0,Y 417.129,Z 549.551,A -85,B 0,C 180,E1 -10175.317,E2 -10175.317} C_VEL
LIN {X 0,Y 417.234,Z 545.461,A -85,B 0,C 180,E1 -10176.771,E2 -10176.771} C_VEL
LIN {X 0,Y 417.54,Z 539.18,A -85,B 0,C 180,E1 -10178.469,E2 -10178.469} C_VEL
LIN {X 0,Y 417.935,Z 532.335,A -85,B 0,C 180,E1 -10179.925,E2 -10179.925} C_VEL
LIN {X 0,Y 418.357,Z 525.347,A -85,B 0,C 180,E1 -10181.139,E2 -10181.139} C_VEL
LIN {X 0,Y 419.015,Z 516.937,A -85,B 0,C 180,E1 -10182.348,E2 -10182.348} C_VEL
LIN {X 0,Y 419.666,Z 506.556,A -85,B 0,C 180,E1 -10183.559,E2 -10183.559} C_VEL
LIN {X 0,Y 420.342,Z 496.278,A -85,B 0,C 180,E1 -10184.524,E2 -10184.524} C_VEL
LIN {X 0,Y 420.985,Z 485.034,A -85,B 0,C 180,E1 -10185.368,E2 -10185.368} C_VEL
LIN {X 0,Y 421.357,Z 475.435,A -85,B 0,C 180,E1 -10185.937,E2 -10185.937} C_VEL
LIN {X 0,Y 419.57,Z 462.455,A -85,B 0,C 180,E1 -10186.591,E2 -10186.591} C_VEL
LIN {X 0,Y 417.497,Z 449.331,A -85,B 0,C 180,E1 -10187.07,E2 -10187.07} C_VEL
LIN {X 0,Y 417.806,Z 440.375,A -85,B 0,C 180,E1 -10191.201,E2 -10191.201} C_VEL
LIN {X 0,Y 418.102,Z 432.721,A -85,B 0,C 180,E1 -10194.81,E2 -10194.81} C_VEL
LIN {X 0,Y 418.496,Z 424.887,A -85,B 0,C 180,E1 -10198.594,E2 -10198.594} C_VEL
LIN {X 0,Y 418.883,Z 419.325,A -85,B 0,C 180,E1 -10201.339,E2 -10201.339} C_VEL
LIN {X 0,Y 419.253,Z 412.619,A -85,B 0,C 180,E1 -10204.775,E2 -10204.775} C_VEL
LIN {X 0,Y 419.222,Z 409.509,A -85,B 0,C 180,E1 -10206.419,E2 -10206.419} C_VEL
LIN {X 0,Y 418.394,Z 403.73,A -85,B 0,C 180,E1 -10209.665,E2 -10209.665} C_VEL
LIN {X 0,Y 418.299,Z 403.381,A -85,B 0,C 180,E1 -10209.989,E2 -10209.989} C_VEL
LIN {X 0,Y 418.264,Z 403.383,A -85,B 0,C 180,E1 -10213.543,E2 -10213.543} C_VEL
LIN {X 0,Y 418.211,Z 403.389,A -85,B 0,C 180,E1 -10216.449,E2 -10216.449} C_VEL
LIN {X 0,Y 418.219,Z 403.391,A -85,B 0,C 180,E1 -10219.129,E2 -10219.129} C_VEL
LIN {X 0,Y 418.229,Z 403.387,A -85,B 0,C 180,E1 -10222.165,E2 -10222.165} C_VEL
LIN {X 0,Y 418.26,Z 403.384,A -85,B 0,C 180,E1 -10225.419,E2 -10225.419} C_VEL
LIN {X 0,Y 418.211,Z 403.393,A -85,B 0,C 180,E1 -10228.604,E2 -10228.604} C_VEL
LIN {X 0,Y 418.288,Z 403.38,A -85,B 0,C 180,E1 -10231.936,E2 -10231.936} C_VEL
LIN {X 0,Y 418.283,Z 403.382,A -85,B 0,C 180,E1 -10235.162,E2 -10235.162} C_VEL
LIN {X 0,Y 418.227,Z 403.39,A -85,B 0,C 180,E1 -10238.303,E2 -10238.303} C_VEL
LIN {X 0,Y 418.276,Z 403.382,A -85,B 0,C 180,E1 -10241.383,E2 -10241.383} C_VEL
LIN {X 0,Y 418.294,Z 403.382,A -85,B 0,C 180,E1 -10244.405,E2 -10244.405} C_VEL
LIN {X 0,Y 418.347,Z 403.373,A -85,B 0,C 180,E1 -10247.385,E2 -10247.385} C_VEL
LIN {X 0,Y 418.333,Z 403.376,A -85,B 0,C 180,E1 -10250.328,E2 -10250.328} C_VEL
LIN {X 0,Y 418.486,Z 403.356,A -85,B 0,C 180,E1 -10253.249,E2 -10253.249} C_VEL
LIN {X 0,Y 418.337,Z 403.375,A -85,B 0,C 180,E1 -10255.181,E2 -10255.181} C_VEL
LIN {X 0,Y 418.536,Z 403.351,A -85,B 0,C 180,E1 -10258.075,E2 -10258.075} C_VEL
LIN {X 0,Y 418.665,Z 403.335,A -85,B 0,C 180,E1 -10260,E2 -10260} C_VEL
LIN {X 0,Y 418.505,Z 403.355,A -85,B 0,C 180,E1 -10262.888,E2 -10262.888} C_VEL
LIN {X 0,Y 418.486,Z 403.357,A -85,B 0,C 180,E1 -10266.751,E2 -10266.751} C_VEL
LIN {X 0,Y 418.334,Z 403.376,A -85,B 0,C 180,E1 -10269.671,E2 -10269.671} C_VEL
LIN {X 0,Y 418.346,Z 403.373,A -85,B 0,C 180,E1 -10273.006,E2 -10273.006} C_VEL
LIN {X 0,Y 418.304,Z 403.379,A -85,B 0,C 180,E1 -10276.736,E2 -10276.736} C_VEL
LIN {X 0,Y 418.263,Z 403.384,A -85,B 0,C 180,E1 -10279.791,E2 -10279.791} C_VEL
LIN {X 0,Y 418.231,Z 403.387,A -85,B 0,C 180,E1 -10282.736,E2 -10282.736} C_VEL
LIN {X 0,Y 418.263,Z 403.386,A -85,B 0,C 180,E1 -10285.904,E2 -10285.904} C_VEL
LIN {X 0,Y 418.267,Z 403.383,A -85,B 0,C 180,E1 -10289.162,E2 -10289.162} C_VEL
LIN {X 0,Y 418.253,Z 403.383,A -85,B 0,C 180,E1 -10292.845,E2 -10292.845} C_VEL
LIN {X 0,Y 418.242,Z 403.386,A -85,B 0,C 180,E1 -10296.239,E2 -10296.239} C_VEL
LIN {X 0,Y 418.26,Z 403.387,A -85,B 0,C 180,E1 -10299.681,E2 -10299.681} C_VEL
LIN {X 0,Y 418.279,Z 403.38,A -85,B 0,C 180,E1 -10302.33,E2 -10302.33} C_VEL
LIN {X 0,Y 418.269,Z 403.382,A -85,B 0,C 180,E1 -10305.115,E2 -10305.115} C_VEL
LIN {X 0,Y 418.288,Z 403.382,A -85,B 0,C 180,E1 -10307.774,E2 -10307.774} C_VEL
LIN {X 0,Y 418.262,Z 403.387,A -85,B 0,C 180,E1 -10311.56,E2 -10311.56} C_VEL
LIN {X 0,Y 418.256,Z 403.386,A -85,B 0,C 180,E1 -10315.16,E2 -10315.16} C_VEL
LIN {X 0,Y 418.243,Z 403.388,A -85,B 0,C 180,E1 -10317.473,E2 -10317.473} C_VEL
LIN {X 0,Y 418.266,Z 403.383,A -85,B 0,C 180,E1 -10320.896,E2 -10320.896} C_VEL
LIN {X 0,Y 418.269,Z 403.381,A -85,B 0,C 180,E1 -10324.097,E2 -10324.097} C_VEL
LIN {X 0,Y 418.209,Z 403.392,A -85,B 0,C 180,E1 -10327.263,E2 -10327.263} C_VEL
LIN {X 0,Y 418.065,Z 403.531,A -85,B 0,C 180,E1 -10329.328,E2 -10329.328} C_VEL
LIN {X 0,Y 417.961,Z 407.53,A -85,B 0,C 180,E1 -10332.383,E2 -10332.383} C_VEL
LIN {X 0,Y 417.841,Z 411.536,A -85,B 0,C 180,E1 -10335.387,E2 -10335.387} C_VEL
LIN {X 0,Y 417.789,Z 415.561,A -85,B 0,C 180,E1 -10338.355,E2 -10338.355} C_VEL
LIN {X 0,Y 417.644,Z 420.991,A -85,B 0,C 180,E1 -10342.264,E2 -10342.264} C_VEL
LIN {X 0,Y 417.587,Z 425.106,A -85,B 0,C 180,E1 -10345.173,E2 -10345.173} C_VEL
LIN {X 0,Y 417.5,Z 427.739,A -85,B 0,C 180,E1 -10347.015,E2 -10347.015} C_VEL
LIN {X 0,Y 420.417,Z 442.946,A -85,B 0,C 180,E1 -10347.65,E2 -10347.65} C_VEL
LIN {X 0,Y 421.823,Z 451.148,A -85,B 0,C 180,E1 -10348.091,E2 -10348.091} C_VEL
LIN {X 0,Y 421.272,Z 463.059,A -85,B 0,C 180,E1 -10348.805,E2 -10348.805} C_VEL
LIN {X 0,Y 420.594,Z 473.899,A -85,B 0,C 180,E1 -10349.641,E2 -10349.641} C_VEL
LIN {X 0,Y 419.883,Z 484.951,A -85,B 0,C 180,E1 -10350.719,E2 -10350.719} C_VEL
LIN {X 0,Y 419.2,Z 494.798,A -85,B 0,C 180,E1 -10351.922,E2 -10351.922} C_VEL
LIN {X 0,Y 418.572,Z 502.886,A -85,B 0,C 180,E1 -10353.128,E2 -10353.128} C_VEL
LIN {X 0,Y 418.021,Z 510.826,A -85,B 0,C 180,E1 -10354.581,E2 -10354.581} C_VEL
LIN {X 0,Y 417.732,Z 516.193,A -85,B 0,C 180,E1 -10355.794,E2 -10355.794} C_VEL
LIN {X 0,Y 417.614,Z 518.974,A -85,B 0,C 180,E1 -10356.528,E2 -10356.528} C_VEL
LIN {X 0,Y 416.78,Z 521.508,A -85,B 0,C 180,E1 -10357.254,E2 -10357.254} C_VEL
LIN {X 0,Y 413.675,Z 525.085,A -85,B 0,C 180,E1 -10358.458,E2 -10358.458} C_VEL
LIN {X 0,Y 410.651,Z 528,A -85,B 0,C 180,E1 -10359.714,E2 -10359.714} C_VEL
LIN {X 0,Y 409.956,Z 529.338,A -85,B 0,C 180,E1 -10360.511,E2 -10360.511} C_VEL
LIN {X 0,Y 409.907,Z 531.42,A -85,B 0,C 180,E1 -10362.236,E2 -10362.236} C_VEL
LIN {X 0,Y 409.782,Z 532.22,A -85,B 0,C 180,E1 -10363.893,E2 -10363.893} C_VEL
LIN {X 0,Y 409.788,Z 532.171,A -85,B 0,C 180,E1 -10364.907,E2 -10364.907} C_VEL
LIN {X 0,Y 409.86,Z 531.456,A -85,B 0,C 180,E1 -10366.209,E2 -10366.209} C_VEL
LIN {X 0,Y 409.952,Z 529.406,A -85,B 0,C 180,E1 -10367.974,E2 -10367.974} C_VEL
LIN {X 0,Y 410.223,Z 526.404,A -85,B 0,C 180,E1 -10369.564,E2 -10369.564} C_VEL
LIN {X 0,Y 410.494,Z 522.477,A -85,B 0,C 180,E1 -10371.072,E2 -10371.072} C_VEL
LIN {X 0,Y 410.936,Z 516.608,A -85,B 0,C 180,E1 -10372.778,E2 -10372.778} C_VEL
LIN {X 0,Y 411.525,Z 509.081,A -85,B 0,C 180,E1 -10374.465,E2 -10374.465} C_VEL
LIN {X 0,Y 412.149,Z 502.114,A -85,B 0,C 180,E1 -10375.72,E2 -10375.72} C_VEL
LIN {X 0,Y 412.899,Z 492.888,A -85,B 0,C 180,E1 -10377.085,E2 -10377.085} C_VEL
LIN {X 0,Y 413.774,Z 483.366,A -85,B 0,C 180,E1 -10378.215,E2 -10378.215} C_VEL
LIN {X 0,Y 414.59,Z 471.99,A -85,B 0,C 180,E1 -10379.306,E2 -10379.306} C_VEL
LIN {X 0,Y 415.437,Z 459.99,A -85,B 0,C 180,E1 -10380.201,E2 -10380.201} C_VEL
LIN {X 0,Y 415.766,Z 451.865,A -85,B 0,C 180,E1 -10380.684,E2 -10380.684} C_VEL
LIN {X 0,Y 413.288,Z 439.389,A -85,B 0,C 180,E1 -10381.406,E2 -10381.406} C_VEL
LIN {X 0,Y 410.348,Z 428.165,A -85,B 0,C 180,E1 -10381.951,E2 -10381.951} C_VEL
LIN {X 0,Y 410.447,Z 423.265,A -85,B 0,C 180,E1 -10385.603,E2 -10385.603} C_VEL
LIN {X 0,Y 410.643,Z 420.029,A -85,B 0,C 180,E1 -10388.069,E2 -10388.069} C_VEL
LIN {X 0,Y 410.821,Z 416.037,A -85,B 0,C 180,E1 -10391.174,E2 -10391.174} C_VEL
LIN {X 0,Y 410.97,Z 411.884,A -85,B 0,C 180,E1 -10394.518,E2 -10394.518} C_VEL
LIN {X 0,Y 411.187,Z 408.532,A -85,B 0,C 180,E1 -10397.302,E2 -10397.302} C_VEL
LIN {X 0,Y 411.244,Z 405.083,A -85,B 0,C 180,E1 -10400.266,E2 -10400.266} C_VEL
LIN {X 0,Y 411.179,Z 404.521,A -85,B 0,C 180,E1 -10400.772,E2 -10400.772} C_VEL
LIN {X 0,Y 411.189,Z 404.272,A -85,B 0,C 180,E1 -10403.447,E2 -10403.447} C_VEL
LIN {X 0,Y 411.203,Z 404.268,A -85,B 0,C 180,E1 -10406.873,E2 -10406.873} C_VEL
LIN {X 0,Y 411.236,Z 404.261,A -85,B 0,C 180,E1 -10410.642,E2 -10410.642} C_VEL
LIN {X 0,Y 411.233,Z 404.261,A -85,B 0,C 180,E1 -10413.619,E2 -10413.619} C_VEL
LIN {X 0,Y 411.191,Z 404.267,A -85,B 0,C 180,E1 -10416.852,E2 -10416.852} C_VEL
LIN {X 0,Y 411.209,Z 404.264,A -85,B 0,C 180,E1 -10420.05,E2 -10420.05} C_VEL
LIN {X 0,Y 411.257,Z 404.257,A -85,B 0,C 180,E1 -10423.131,E2 -10423.131} C_VEL
LIN {X 0,Y 411.299,Z 404.251,A -85,B 0,C 180,E1 -10426.896,E2 -10426.896} C_VEL
LIN {X 0,Y 411.288,Z 404.252,A -85,B 0,C 180,E1 -10430.161,E2 -10430.161} C_VEL
LIN {X 0,Y 411.454,Z 404.233,A -85,B 0,C 180,E1 -10433.133,E2 -10433.133} C_VEL
LIN {X 0,Y 411.305,Z 404.253,A -85,B 0,C 180,E1 -10435.099,E2 -10435.099} C_VEL
LIN {X 0,Y 411.508,Z 404.229,A -85,B 0,C 180,E1 -10438.043,E2 -10438.043} C_VEL
LIN {X 0,Y 411.636,Z 404.21,A -85,B 0,C 180,E1 -10440,E2 -10440} C_VEL
LIN {X 0,Y 411.462,Z 404.232,A -85,B 0,C 180,E1 -10442.937,E2 -10442.937} C_VEL
LIN {X 0,Y 411.455,Z 404.232,A -85,B 0,C 180,E1 -10446.867,E2 -10446.867} C_VEL
LIN {X 0,Y 411.303,Z 404.254,A -85,B 0,C 180,E1 -10449.839,E2 -10449.839} C_VEL
LIN {X 0,Y 411.309,Z 404.253,A -85,B 0,C 180,E1 -10453.11,E2 -10453.11} C_VEL
LIN {X 0,Y 411.259,Z 404.258,A -85,B 0,C 180,E1 -10456.87,E2 -10456.87} C_VEL
LIN {X 0,Y 411.226,Z 404.263,A -85,B 0,C 180,E1 -10459.987,E2 -10459.987} C_VEL
LIN {X 0,Y 411.199,Z 404.267,A -85,B 0,C 180,E1 -10463.148,E2 -10463.148} C_VEL
LIN {X 0,Y 411.234,Z 404.265,A -85,B 0,C 180,E1 -10466.381,E2 -10466.381} C_VEL
LIN {X 0,Y 411.207,Z 404.265,A -85,B 0,C 180,E1 -10469.712,E2 -10469.712} C_VEL
LIN {X 0,Y 411.203,Z 404.264,A -85,B 0,C 180,E1 -10473.156,E2 -10473.156} C_VEL
LIN {X 0,Y 411.192,Z 404.264,A -85,B 0,C 180,E1 -10476.554,E2 -10476.554} C_VEL
